	W =    47.745 deg,	P =     8.599 deg,	R =   -35.895 deg
   GP2:
	UF : 1, UT : 1,
	J1=     0.000 deg,	J2=   180.000 deg
};
P[182]{
   GP1:
	UF : 1, UT : 1,		CONFIG : 'N U T, 0, 0, 0',
	X =  2150.796  mm,	Y =    51.228  mm,	Z =   379.826  mm,
	W =     9.396 deg,	P =    -3.028 deg,	R =   -24.284 deg
   GP2:
	UF : 1, UT : 1,
	J1=     0.000 deg,	J2=   180.000 deg
};
P[183]{
   GP1:
	UF : 1, UT : 1,		CONFIG : 'N U T, 0, 0, 0',
	X =  1058.698  mm,	Y =   195.065  mm,	Z =  1283.367  mm,
	W =    73.635 deg,	P =    26.735 deg,	R =   -73.196 deg
   GP2:
	UF : 1, UT : 1,
	J1=   -90.000 deg,	J2=   -90.000 deg
};
P[184]{
   GP1:
	UF : 1, UT : 1,		CONFIG : 'N U T, 0, 0, 0',
	X =  2161.838  mm,	Y =  -354.344  mm,	Z =   373.103  mm,
	W =   -42.503 deg,	P =    -2.383 deg,	R =   -32.742 deg
   GP2:
	UF : 1, UT : 1,
	J1=     0.000 deg,	J2=   180.000 deg
};
P[185]{
   GP1:
	UF : 1, UT : 1,		CONFIG : 'N U T, 0, 0, 0',
	X =  2732.660  mm,	Y =  -291.498  mm,	Z =   459.463  mm,
	W =    29.147 deg,	P =    30.453 deg,	R =  -132.266 deg
   GP2:
	UF : 1, UT : 1,
	J1=    90.000 deg,	J2=     0.000 deg
};
P[186]{
   GP1:
	UF : 1, UT : 1,		CONFIG : 'N U T, 0, 0, 1',
	X =  2737.828  mm,	Y =  -335.614  mm,	Z =   459.309  mm,
	W =    29.459 deg,	P =    30.697 deg,	R =  -132.107 deg
   GP2:
	UF : 1, UT : 1,
	J1=    90.000 deg,	J2=     0.000 deg
};
P[187]{
   GP1:
	UF : 1, UT : 1,		CONFIG : 'N U T, 0, 0, 1',
	X =  2748.682  mm,	Y =  -359.447  mm,	Z =   458.247  mm,
	W =    32.708 deg,	P =    26.756 deg,	R =  -103.211 deg
   GP2:
	UF : 1, UT : 1,
	J1=    90.000 deg,	J2=     0.000 deg
};
P[188]{
   GP1:
	UF : 1, UT : 1,		CONFIG : 'N U T, 0, 0, 1',
	X =  2782.788  mm,	Y =  -368.053  mm,	Z =   461.277  mm,
	W =    32.871 deg,	P =    19.630 deg,	R =   -83.146 deg
   GP2:
	UF : 1, UT : 1,
	J1=    90.000 deg,	J2=     0.000 deg
};
P[189]{
   GP1:
	UF : 1, UT : 1,		CONFIG : 'N U T, 0, 0, 0',
	X =  2149.286  mm,	Y =  -279.133  mm,	Z =   456.472  mm,
	W =   -44.186 deg,	P =    -9.562 deg,	R =     3.909 deg
   GP2:
	UF : 1, UT : 1,
	J1=     0.000 deg,	J2=   180.000 deg
};
P[190]{
   GP1:
	UF : 1, UT : 1,		CONFIG : 'N U T, 0, 0, 1',
	X =  1982.724  mm,	Y =   -25.313  mm,	Z =   235.548  mm,
	W =    21.889 deg,	P =    35.316 deg,	R =  -145.925 deg
   GP2:
	UF : 1, UT : 1,
	J1=     0.000 deg,	J2=   180.000 deg
};
P[191]{
   GP1:
	UF : 1, UT : 1,		CONFIG : 'N U T, 0, 0, 1',
	X =  2182.725  mm,	Y =  -216.312  mm,	Z =    -6.136  mm,
	W =    32.857 deg,	P =    25.665 deg,	R =  -124.570 deg
   GP2:
	UF : 1, UT : 1,
	J1=     0.000 deg,	J2=   180.000 deg
};
P[192]{
   GP1:
	UF : 1, UT : 1,		CONFIG : 'N U T, 0, 0, 0',
	X =  2740.807  mm,	Y =   282.456  mm,	Z =   454.339  mm,
	W =   -36.614 deg,	P =    28.247 deg,	R =   122.490 deg
   GP2:
	UF : 1, UT : 1,
	J1=    90.000 deg,	J2=     0.000 deg
};
P[193]{
   GP1:
	UF : 1, UT : 1,		CONFIG : 'N U T, 0, 0, 0',
	X =  2740.471  mm,	Y =   330.671  mm,	Z =   455.272  mm,
	W =   -36.614 deg,	P =    28.247 deg,	R =   122.490 deg
   GP2:
	UF : 1, UT : 1,
	J1=    90.000 deg,	J2=     0.000 deg
};
P[194]{
   GP1:
	UF : 1, UT : 1,		CONFIG : 'N U T, 0, 0, 0',
	X =  2760.137  mm,	Y =   356.906  mm,	Z =   456.179  mm,
	W =   -32.204 deg,	P =    27.169 deg,	R =   100.051 deg
   GP2:
	UF : 1, UT : 1,
	J1=    90.000 deg,	J2=     0.000 deg
};
P[195]{
   GP1:
	UF : 1, UT : 1,		CONFIG : 'N U T, 0, 0, 1',
	X =  2185.038  mm,	Y =   -47.631  mm,	Z =   -82.880  mm,
	W =     1.218 deg,	P =    44.987 deg,	R =  -147.433 deg
   GP2:
	UF : 1, UT : 1,
	J1=     0.000 deg,	J2=   180.000 deg
};
P[196]{
   GP1:
	UF : 1, UT : 1,		CONFIG : 'N U T, 0, 0, 0',
	X =  2185.038  mm,	Y =   213.369  mm,	Z =   -82.880  mm,
	W =   -26.253 deg,	P =    37.378 deg,	R =   139.534 deg
   GP2:
	UF : 1, UT : 1,
	J1=     0.000 deg,	J2=   180.000 deg
};
P[197]{
   GP1:
	UF : 1, UT : 1,		CONFIG : 'N U T, 0, 0, 0',
	X =  2776.222  mm,	Y =   360.760  mm,	Z =   461.623  mm,
	W =   -28.646 deg,	P =    22.121 deg,	R =    94.724 deg
   GP2:
	UF : 1, UT : 1,
	J1=    90.000 deg,	J2=     0.000 deg
};
P[198]{
   GP1:
	UF : 1, UT : 1,		CONFIG : 'N U T, 0, 0, 0',
	X =  1666.073  mm,	Y =   232.940  mm,	Z =   357.763  mm,
	W =    31.327 deg,	P =    33.496 deg,	R =    49.952 deg
   GP2:
	UF : 1, UT : 1,
	J1=    90.000 deg,	J2=     0.000 deg
};
P[199]{
   GP1:
	UF : 1, UT : 1,		CONFIG : 'N U T, 0, 0, 0',
	X =  1669.367  mm,	Y =   161.118  mm,	Z =   359.810  mm,
	W =    31.331 deg,	P =    33.498 deg,	R =    49.952 deg
   GP2:
	UF : 1, UT : 1,
	J1=    90.000 deg,	J2=     0.000 deg
};
P[200]{
   GP1:
	UF : 1, UT : 1,		CONFIG : 'N U T, 0, 0, 0',
	X =  2149.428  mm,	Y =    61.346  mm,	Z =   -40.697  mm,
	W =    14.710 deg,	P =    43.024 deg,	R =   172.922 deg
   GP2:
	UF : 1, UT : 1,
	J1=     0.000 deg,	J2=   180.000 deg
};
P[201]{
   GP1:
	UF : 1, UT : 1,		CONFIG : 'N U T, 0, 0, 0',
	X =  1379.179  mm,	Y =     5.048  mm,	Z =   295.119  mm,
	W =    -2.053 deg,	P =    45.296 deg,	R =  -168.776 deg
   GP2:
	UF : 1, UT : 1,
	J1=     0.000 deg,	J2=   180.000 deg
};
P[202]{
   GP1:
	UF : 1, UT : 1,		CONFIG : 'N U T, 0, 0, 1',
	X =  1381.432  mm,	Y =  -574.038  mm,	Z =   156.436  mm,
	W =    42.351 deg,	P =    16.902 deg,	R =  -106.783 deg
   GP2:
	UF : 1, UT : 1,
	J1=     0.000 deg,	J2=   180.000 deg
};
P[203]{
   GP1:
	UF : 1, UT : 1,		CONFIG : 'N U T, 0, 0, 0',
	X =  1672.296  mm,	Y =  -245.157  mm,	Z =   359.474  mm,
	W =   -34.074 deg,	P =    31.387 deg,	R =   -56.109 deg
   GP2:
	UF : 1, UT : 1,
	J1=    90.000 deg,	J2=     0.000 deg
};
P[204]{
   GP1:
	UF : 1, UT : 1,		CONFIG : 'N U T, 0, 0, 0',
	X =  1674.067  mm,	Y =  -171.272  mm,	Z =   358.368  mm,
	W =   -34.074 deg,	P =    31.387 deg,	R =   -56.109 deg
   GP2:
	UF : 1, UT : 1,
	J1=    90.000 deg,	J2=     0.000 deg
};
P[205]{
   GP1:
	UF : 1, UT : 1,		CONFIG : 'N U T, 0, 0, 0',
	X =  1806.951  mm,	Y =  -401.301  mm,	Z =   820.124  mm,
	W =     -.611 deg,	P =      .925 deg,	R =   -33.342 deg
   GP2:
	UF : 1, UT : 1,
	J1=    45.000 deg,	J2=     0.000 deg
};
P[206]{
   GP1:
	UF : 1, UT : 1,		CONFIG : 'N U T, 0, 0, 1',
	X =  1351.612  mm,	Y =  -644.118  mm,	Z =   196.361  mm,
	W =    42.489 deg,	P =    16.481 deg,	R =  -107.209 deg
   GP2:
	UF : 1, UT : 1,
	J1=     0.000 deg,	J2=   180.000 deg
};
P[207]{
   GP1:
	UF : 1, UT : 1,		CONFIG : 'N U T, 0, 0, 0',
	X =  1351.612  mm,	Y =     1.774  mm,	Z =   196.362  mm,
	W =     -.786 deg,	P =    44.995 deg,	R =   178.888 deg
   GP2:
	UF : 1, UT : 1,
	J1=     0.000 deg,	J2=   180.000 deg
};
P[208]{
   GP1:
	UF : 1, UT : 1,		CONFIG : 'N U T, 0, 0, 0',
	X =  1811.177  mm,	Y =  -171.928  mm,	Z =   822.372  mm,
	W =     -.615 deg,	P =      .929 deg,	R =   -33.344 deg
   GP2:
	UF : 1, UT : 1,
	J1=    45.000 deg,	J2=     0.000 deg
};
P[209]{
   GP1:
	UF : 1, UT : 1,		CONFIG : 'N U T, 0, 0, 0',
	X =  1807.900  mm,	Y =   392.843  mm,	Z =   821.281  mm,
	W =     -.607 deg,	P =      .924 deg,	R =    40.442 deg
   GP2:
	UF : 1, UT : 1,
	J1=    45.000 deg,	J2=     0.000 deg
};
P[210]{
   GP1:
	UF : 1, UT : 1,		CONFIG : 'N U T, 0, 0, 0',
	X =  1404.034  mm,	Y =  -379.314  mm,	Z =   119.254  mm,
	W =    18.566 deg,	P =    41.762 deg,	R =  -153.239 deg
   GP2:
	UF : 1, UT : 1,
	J1=     0.000 deg,	J2=   180.000 deg
};
P[211]{
   GP1:
	UF : 1, UT : 1,		CONFIG : 'N U T, 0, 0, 0',
	X =  1404.034  mm,	Y =   331.497  mm,	Z =   119.254  mm,
	W =   -20.958 deg,	P =    40.782 deg,	R =   149.612 deg
   GP2:
	UF : 1, UT : 1,
	J1=     0.000 deg,	J2=   180.000 deg
};
P[212]{
   GP1:
	UF : 1, UT : 1,		CONFIG : 'N U T, 0, 0, 0',
	X =  1805.706  mm,	Y =   162.058  mm,	Z =   821.772  mm,
	W =     -.607 deg,	P =      .924 deg,	R =    40.442 deg
   GP2:
	UF : 1, UT : 1,
	J1=    45.000 deg,	J2=     0.000 deg
};
P[213]{
   GP1:
	UF : 1, UT : 1,		CONFIG : 'N U T, 0, 0, 0',
	X =  2179.485  mm,	Y =   641.712  mm,	Z =  1313.269  mm,
	W =     -.150 deg,	P =     3.186 deg,	R =     -.120 deg
   GP2:
	UF : 1, UT : 1,
	J1=   124.996 deg,	J2=     0.000 deg
};
P[214]{
   GP1:
	UF : 1, UT : 1,		CONFIG : 'N U T, 0, 0, 0',
	X =  1267.764  mm,	Y =    -5.079  mm,	Z =   257.741  mm,
	W =     -.786 deg,	P =    44.995 deg,	R =   178.888 deg
   GP2:
	UF : 1, UT : 1,
	J1=     0.000 deg,	J2=   180.000 deg
};
P[215]{
   GP1:
	UF : 1, UT : 1,		CONFIG : 'N U T, 0, 0, 0',
	X =  1267.763  mm,	Y =   567.064  mm,	Z =   257.741  mm,
	W =    24.666 deg,	P =    38.913 deg,	R =  -143.830 deg
   GP2:
	UF : 1, UT : 1,
	J1=     0.000 deg,	J2=   180.000 deg
};
P[216]{
   GP1:
	UF : 1, UT : 1,		CONFIG : 'N U T, 0, 0, 0',
	X =  2180.448  mm,	Y =   484.330  mm,	Z =  1313.381  mm,
	W =      .050 deg,	P =     3.285 deg,	R =     -.057 deg
   GP2:
	UF : 1, UT : 1,
	J1=   124.995 deg,	J2=     0.000 deg
};
P[217]{
   GP1:
	UF : 1, UT : 1,		CONFIG : 'N U T, 0, 0, 0',
	X =  2180.629  mm,	Y =   441.870  mm,	Z =  1314.110  mm,
	W =   -10.967 deg,	P =     3.763 deg,	R =     -.257 deg
   GP2:
	UF : 1, UT : 1,
	J1=   124.999 deg,	J2=     0.000 deg
};
P[218]{
   GP1:
	UF : 1, UT : 1,		CONFIG : 'N U T, 0, 0, 0',
	X =  2166.448  mm,	Y =     9.539  mm,	Z =  1331.644  mm,
	W =     -.712 deg,	P =     8.094 deg,	R =     -.112 deg
   GP2:
	UF : 1, UT : 1,
	J1=   124.996 deg,	J2=     0.000 deg
};
P[219]{
   GP1:
	UF : 1, UT : 1,		CONFIG : 'N U T, 0, 0, 0',
	X =  1302.181  mm,	Y =   638.659  mm,	Z =   248.465  mm,
	W =    31.136 deg,	P =    34.298 deg,	R =  -133.008 deg
   GP2:
	UF : 1, UT : 1,
	J1=     0.000 deg,	J2=   180.000 deg
};
P[220]{
   GP1:
	UF : 1, UT : 1,		CONFIG : 'N U T, 0, 0, 0',
	X =  1186.272  mm,	Y =   472.511  mm,	Z =   672.833  mm,
	W =    32.440 deg,	P =    45.276 deg,	R =   -70.624 deg
   GP2:
	UF : 1, UT : 1,
	J1=     0.000 deg,	J2=   180.000 deg
};
P[221]{
   GP1:
	UF : 1, UT : 1,		CONFIG : 'N U T, 0, 0, 0',
	X =  2166.019  mm,	Y =  -184.522  mm,	Z =  1332.900  mm,
	W =     -.016 deg,	P =    10.106 deg,	R =      .980 deg
   GP2:
	UF : 1, UT : 1,
	J1=   125.000 deg,	J2=     0.000 deg
};
P[222]{
   GP1:
	UF : 1, UT : 1,		CONFIG : 'N U T, 0, 0, 0',
	X =  2166.456  mm,	Y =  -407.129  mm,	Z =  1331.643  mm,
	W =     -.927 deg,	P =     7.509 deg,	R =     -.098 deg
   GP2:
	UF : 1, UT : 1,
	J1=   125.000 deg,	J2=     0.000 deg
};
P[223]{
   GP1:
	UF : 1, UT : 1,		CONFIG : 'N U T, 0, 0, 0',
	X =  2167.632  mm,	Y =   399.347  mm,	Z =  1331.502  mm,
	W =      .164 deg,	P =     6.215 deg,	R =      .006 deg
   GP2:
	UF : 1, UT : 1,
	J1=   125.000 deg,	J2=     0.000 deg
};
P[224]{
   GP1:
	UF : 1, UT : 1,		CONFIG : 'N U T, 0, 0, 0',
	X =  1759.654  mm,	Y =  1128.978  mm,	Z =   266.859  mm,
	W =   -16.763 deg,	P =    16.253 deg,	R =    47.184 deg
   GP2:
	UF : 1, UT : 1,
	J1=    90.000 deg,	J2=    90.000 deg
};
P[225]{
   GP1:
	UF : 1, UT : 1,		CONFIG : 'N U T, 0, 0, 0',
	X =  1547.891  mm,	Y =   -77.836  mm,	Z =    80.464  mm,
	W =     5.459 deg,	P =    -9.689 deg,	R =   -27.215 deg
   GP2:
	UF : 1, UT : 1,
	J1=     0.000 deg,	J2=   180.000 deg
};
P[226]{
   GP1:
	UF : 1, UT : 1,		CONFIG : 'N U T, 0, 0, 0',
	X =  2166.862  mm,	Y =   175.690  mm,	Z =  1332.608  mm,
	W =      .990 deg,	P =     7.423 deg,	R =      .117 deg
   GP2:
	UF : 1, UT : 1,
	J1=   125.000 deg,	J2=     0.000 deg
};
P[227]{
   GP1:
	UF : 1, UT : 1,		CONFIG : 'N U T, 0, 0, 0',
	X =  2166.171  mm,	Y =     8.099  mm,	Z =  1332.684  mm,
	W =    -1.725 deg,	P =     7.606 deg,	R =     2.359 deg
   GP2:
	UF : 1, UT : 1,
	J1=   125.000 deg,	J2=     0.000 deg
};
P[228]{
   GP1:
	UF : 1, UT : 1,		CONFIG : 'N U T, 0, 0, 0',
	X =  2179.486  mm,	Y =  -651.866  mm,	Z =  1318.869  mm,
	W =      .005 deg,	P =     8.099 deg,	R =      .006 deg
   GP2:
	UF : 1, UT : 1,
	J1=   125.000 deg,	J2=     0.000 deg
};
P[229]{
   GP1:
	UF : 1, UT : 1,		CONFIG : 'N U T, 0, 0, 0',
	X =  2179.374  mm,	Y =  -454.527  mm,	Z =  1315.208  mm,
	W =      .023 deg,	P =     7.896 deg,	R =     -.019 deg
   GP2:
	UF : 1, UT : 1,
	J1=   125.000 deg,	J2=     0.000 deg
};
P[230]{
   GP1:
	UF : 1, UT : 1,		CONFIG : 'N U T, 0, 0, 0',
	X =  1458.812  mm,	Y =  -160.809  mm,	Z =   231.788  mm,
	W =     9.627 deg,	P =   -18.262 deg,	R =   -28.428 deg
   GP2:
	UF : 1, UT : 1,
	J1=     0.000 deg,	J2=   180.000 deg
};
P[231]{
   GP1:
	UF : 1, UT : 1,		CONFIG : 'N U T, 0, 0, 0',
	X =  2179.713  mm,	Y =  -448.929  mm,	Z =  1315.415  mm,
	W =     8.588 deg,	P =     5.688 deg,	R =      .847 deg
   GP2:
	UF : 1, UT : 1,
	J1=   125.000 deg,	J2=     0.000 deg
};
P[232]{
   GP1:
	UF : 1, UT : 1,		CONFIG : 'N U T, 0, 0, 0',
	X =  2140.306  mm,	Y =   407.443  mm,	Z =   274.579  mm,
	W =    39.266 deg,	P =    23.844 deg,	R =     9.200 deg
   GP2:
	UF : 1, UT : 1,
	J1=     0.000 deg,	J2=   180.000 deg
};
P[233]{
   GP1:
	UF : 1, UT : 1,		CONFIG : 'N U T, 0, 0, 0',
	X =  2171.990  mm,	Y =   -24.925  mm,	Z =  -336.558  mm,
	W =    -4.854 deg,	P =     4.648 deg,	R =    10.738 deg
   GP2:
	UF : 1, UT : 1,
	J1=    45.000 deg,	J2=   182.246 deg
};
P[234]{
   GP1:
	UF : 1, UT : 1,		CONFIG : 'N U T, 0, 0, 0',
	X =  2525.957  mm,	Y =  -153.860  mm,	Z =   104.179  mm,
	W =    36.503 deg,	P =    18.679 deg,	R =   -19.970 deg
   GP2:
	UF : 1, UT : 1,
	J1=    80.000 deg,	J2=    90.000 deg
};
P[235]{
   GP1:
	UF : 1, UT : 1,		CONFIG : 'N U T, 0, 0, 0',
	X =  2443.957  mm,	Y =  -153.860  mm,	Z =    41.179  mm,
	W =    36.503 deg,	P =    18.679 deg,	R =    32.647 deg
   GP2:
	UF : 1, UT : 1,
	J1=    80.000 deg,	J2=    90.000 deg
};
P[236]{
   GP1:
	UF : 1, UT : 1,		CONFIG : 'N U T, 0, 0, 0',
	X =  2156.848  mm,	Y =   408.546  mm,	Z =   273.021  mm,
	W =    39.276 deg,	P =    23.852 deg,	R =   -24.752 deg
   GP2:
	UF : 1, UT : 1,
	J1=     0.000 deg,	J2=   180.000 deg
};
P[237]{
   GP1:
	UF : 1, UT : 1,		CONFIG : 'N U T, 0, 0, 0',
	X =  2192.264  mm,	Y =   408.269  mm,	Z =   272.683  mm,
	W =    39.348 deg,	P =    23.574 deg,	R =   -24.954 deg
   GP2:
	UF : 1, UT : 1,
	J1=     0.000 deg,	J2=   180.000 deg
};
P[238]{
   GP1:
	UF : 1, UT : 1,		CONFIG : 'N U T, 0, 0, 0',
	X =  2195.713  mm,	Y =   409.133  mm,	Z =   275.050  mm,
	W =    41.358 deg,	P =    16.787 deg,	R =   -30.152 deg
   GP2:
	UF : 1, UT : 1,
	J1=     0.000 deg,	J2=   180.000 deg
};
P[239]{
   GP1:
	UF : 1, UT : 1,		CONFIG : 'N U T, 0, 0, 0',
	X =  2131.308  mm,	Y =  -414.633  mm,	Z =   275.688  mm,
	W =   -42.902 deg,	P =    -2.083 deg,	R =   -37.986 deg
   GP2:
	UF : 1, UT : 1,
	J1=     0.000 deg,	J2=   180.000 deg
};
P[240]{
   GP1:
	UF : 1, UT : 1,		CONFIG : 'N U T, 0, 0, 0',
	X =  2443.958  mm,	Y =  -141.290  mm,	Z =    41.179  mm,
	W =    36.502 deg,	P =    18.679 deg,	R =    44.252 deg
   GP2:
	UF : 1, UT : 1,
	J1=    80.000 deg,	J2=    90.000 deg
};
P[241]{
   GP1:
	UF : 1, UT : 1,		CONFIG : 'N U T, 0, 0, 0',
	X =  2525.957  mm,	Y =  -153.860  mm,	Z =   104.179  mm,
	W =    36.503 deg,	P =    18.679 deg,	R =   -19.970 deg
   GP2:
	UF : 1, UT : 1,
	J1=    80.000 deg,	J2=    90.000 deg
};
P[242]{
   GP1:
	UF : 1, UT : 1,		CONFIG : 'N U T, 0, 0, 0',
	X =  1638.942  mm,	Y =  -220.932  mm,	Z =   176.092  mm,
	W =    39.659 deg,	P =    20.135 deg,	R =   -30.806 deg
   GP2:
	UF : 1, UT : 1,
	J1=    90.000 deg,	J2=    90.000 deg
};
P[243]{
   GP1:
	UF : 1, UT : 1,		CONFIG : 'N U T, 0, 0, 0',
	X =  1677.355  mm,	Y =  -241.647  mm,	Z =    77.021  mm,
	W =    39.659 deg,	P =    20.135 deg,	R =   -14.061 deg
   GP2:
	UF : 1, UT : 1,
	J1=    90.000 deg,	J2=    90.000 deg
};
P[244]{
   GP1:
	UF : 1, UT : 1,		CONFIG : 'N U T, 0, 0, 0',
	X =  2148.323  mm,	Y =  -414.723  mm,	Z =   274.084  mm,
	W =   -42.900 deg,	P =    -2.086 deg,	R =    -3.516 deg
   GP2:
	UF : 1, UT : 1,
	J1=     0.000 deg,	J2=   180.000 deg
};
P[245]{
   GP1:
	UF : 1, UT : 1,		CONFIG : 'N U T, 0, 0, 0',
	X =  2197.502  mm,	Y =  -415.369  mm,	Z =   273.507  mm,
	W =   -42.900 deg,	P =    -2.086 deg,	R =    -3.516 deg
   GP2:
	UF : 1, UT : 1,
	J1=     0.000 deg,	J2=   180.000 deg
};
P[246]{
   GP1:
	UF : 1, UT : 1,		CONFIG : 'N U T, 0, 0, 0',
	X =  2205.828  mm,	Y =  -413.909  mm,	Z =   275.461  mm,
	W =   -37.675 deg,	P =   -22.312 deg,	R =     8.930 deg
   GP2:
	UF : 1, UT : 1,
	J1=     0.000 deg,	J2=   180.000 deg
};
P[247]{
   GP1:
	UF : 1, UT : 1,		CONFIG : 'N U T, 0, 0, 1',
	X =  2230.692  mm,	Y =  -244.712  mm,	Z =  -195.164  mm,
	W =    34.818 deg,	P =    27.072 deg,	R =  -123.443 deg
   GP2:
	UF : 1, UT : 1,
	J1=     0.000 deg,	J2=   180.000 deg
};
P[248]{
   GP1:
	UF : 1, UT : 1,		CONFIG : 'N U T, 0, 0, 0',
	X =  1961.011  mm,	Y =  -250.911  mm,	Z =    63.963  mm,
	W =    38.570 deg,	P =    15.643 deg,	R =   -37.733 deg
   GP2:
	UF : 1, UT : 1,
	J1=    90.000 deg,	J2=    90.000 deg
};
P[249]{
   GP1:
	UF : 1, UT : 1,		CONFIG : 'N U T, 0, 0, 0',
	X =  2227.011  mm,	Y =   -35.911  mm,	Z =    63.963  mm,
	W =    41.142 deg,	P =     1.290 deg,	R =    -4.650 deg
   GP2:
	UF : 1, UT : 1,
	J1=    90.000 deg,	J2=    90.000 deg
};
P[250]{
   GP1:
	UF : 1, UT : 1,		CONFIG : 'N U T, 0, 0, 1',
	X =  2231.573  mm,	Y =   -26.230  mm,	Z =  -195.203  mm,
	W =    34.826 deg,	P =    27.077 deg,	R =  -123.454 deg
   GP2:
	UF : 1, UT : 1,
	J1=     0.000 deg,	J2=   180.000 deg
};
P[251]{
   GP1:
	UF : 1, UT : 1,		CONFIG : 'N U T, 0, 0, 1',
	X =  2228.732  mm,	Y =    -5.925  mm,	Z =  -190.893  mm,
	W =    33.017 deg,	P =    26.717 deg,	R =   -93.421 deg
   GP2:
	UF : 1, UT : 1,
	J1=     0.000 deg,	J2=   180.000 deg
};
P[252]{
   GP1:
	UF : 1, UT : 1,		CONFIG : 'N U T, 0, 0, 0',
	X =  2193.552  mm,	Y =   -35.911  mm,	Z =    63.963  mm,
	W =    41.142 deg,	P =     1.290 deg,	R =    -4.650 deg
   GP2:
	UF : 1, UT : 1,
	J1=    90.000 deg,	J2=    90.000 deg
};
P[253]{
   GP1:
	UF : 1, UT : 1,		CONFIG : 'N U T, 0, 0, 0',
	X =  2230.608  mm,	Y =   237.638  mm,	Z =  -198.866  mm,
	W =   -26.756 deg,	P =    37.336 deg,	R =   139.554 deg
   GP2:
	UF : 1, UT : 1,
	J1=     0.000 deg,	J2=   180.000 deg
};
P[254]{
   GP1:
	UF : 1, UT : 1,		CONFIG : 'N U T, 0, 0, 0',
	X =  2230.167  mm,	Y =    15.957  mm,	Z =  -196.509  mm,
	W =   -26.754 deg,	P =    37.334 deg,	R =   139.553 deg
   GP2:
	UF : 1, UT : 1,
	J1=     0.000 deg,	J2=   180.000 deg
};
P[255]{
   GP1:
	UF : 1, UT : 1,		CONFIG : 'N U T, 0, 0, 0',
	X =  2229.296  mm,	Y =    -3.861  mm,	Z =  -195.798  mm,
	W =   -20.120 deg,	P =    35.519 deg,	R =   111.508 deg
   GP2:
	UF : 1, UT : 1,
	J1=     0.000 deg,	J2=   180.000 deg
};
P[256]{
   GP1:
	UF : 1, UT : 1,		CONFIG : 'N U T, 0, 0, 0',
	X =  2104.646  mm,	Y =   -14.305  mm,	Z =    58.276  mm,
	W =    44.920 deg,	P =     3.025 deg,	R =    -3.029 deg
   GP2:
	UF : 1, UT : 1,
	J1=    90.000 deg,	J2=    90.000 deg
};
P[257]{
   GP1:
	UF : 1, UT : 1,		CONFIG : 'N U T, 0, 0, 0',
	X =  1481.773  mm,	Y =  -649.516  mm,	Z =     4.672  mm,
	W =    42.305 deg,	P =    16.820 deg,	R =  -100.938 deg
   GP2:
	UF : 1, UT : 1,
	J1=     0.000 deg,	J2=   180.000 deg
};
P[258]{
   GP1:
	UF : 1, UT : 1,		CONFIG : 'N U T, 0, 0, 0',
	X =  1483.359  mm,	Y =  -463.806  mm,	Z =     3.440  mm,
	W =    42.353 deg,	P =    16.915 deg,	R =  -100.930 deg
   GP2:
	UF : 1, UT : 1,
	J1=     0.000 deg,	J2=   180.000 deg
};
P[259]{
   GP1:
	UF : 1, UT : 1,		CONFIG : 'N U T, 0, 0, 1',
	X =  1480.083  mm,	Y =  -453.844  mm,	Z =     3.901  mm,
	W =    42.350 deg,	P =    16.901 deg,	R =   -86.937 deg
   GP2:
	UF : 1, UT : 1,
	J1=     0.000 deg,	J2=   180.000 deg
};
P[260]{
   GP1:
	UF : 1, UT : 1,		CONFIG : 'N U T, 0, 0, 0',
	X =  2104.646  mm,	Y =   -54.652  mm,	Z =   175.276  mm,
	W =    44.920 deg,	P =     3.025 deg,	R =    -3.029 deg
   GP2:
	UF : 1, UT : 1,
	J1=    90.000 deg,	J2=    90.000 deg
};
P[261]{
   GP1:
	UF : 1, UT : 1,		CONFIG : 'N U T, 0, 0, 0',
	X =  1705.582  mm,	Y =   -41.652  mm,	Z =   107.776  mm,
	W =    44.920 deg,	P =     3.025 deg,	R =    11.940 deg
   GP2:
	UF : 1, UT : 1,
	J1=    90.000 deg,	J2=    90.000 deg
};
P[262]{
   GP1:
	UF : 1, UT : 1,		CONFIG : 'N U T, 0, 0, -1',
	X =  1457.610  mm,	Y =    -5.074  mm,	Z =    -1.334  mm,
	W =      .944 deg,	P =    42.924 deg,	R =   177.949 deg
   GP2:
	UF : 1, UT : 1,
	J1=     0.000 deg,	J2=   180.000 deg
};
P[263]{
   GP1:
	UF : 1, UT : 1,		CONFIG : 'N U T, 0, 0, 0',
	X =  1456.823  mm,	Y =  -333.215  mm,	Z =     -.642  mm,
	W =    -1.375 deg,	P =    43.930 deg,	R =   175.836 deg
   GP2:
	UF : 1, UT : 1,
	J1=     0.000 deg,	J2=   180.000 deg
};
P[264]{
   GP1:
	UF : 1, UT : 1,		CONFIG : 'N U T, 0, 0, 0',
	X =  1457.144  mm,	Y =  -389.993  mm,	Z =      .340  mm,
	W =     5.164 deg,	P =    43.292 deg,	R =  -179.576 deg
   GP2:
	UF : 1, UT : 1,
	J1=     0.000 deg,	J2=   180.000 deg
};
P[265]{
   GP1:
	UF : 1, UT : 1,		CONFIG : 'N U T, 0, 0, 0',
	X =  1700.208  mm,	Y =   -40.379  mm,	Z =   119.303  mm,
	W =    53.172 deg,	P =     1.611 deg,	R =    24.177 deg
   GP2:
	UF : 1, UT : 1,
	J1=    90.000 deg,	J2=    90.000 deg
};
P[266]{
   GP1:
	UF : 1, UT : 1,		CONFIG : 'N U T, 0, 0, -1',
	X =  1452.091  mm,	Y =   380.184  mm,	Z =     1.132  mm,
	W =    -1.242 deg,	P =    44.316 deg,	R =   179.193 deg
   GP2:
	UF : 1, UT : 1,
	J1=     0.000 deg,	J2=   180.000 deg
};
P[267]{
   GP1:
	UF : 1, UT : 1,		CONFIG : 'N U T, 0, 0, 0',
	X =  1459.905  mm,	Y =    -8.182  mm,	Z =     -.258  mm,
	W =     -.052 deg,	P =    43.981 deg,	R =  -179.147 deg
   GP2:
	UF : 1, UT : 1,
	J1=     0.000 deg,	J2=   180.000 deg
};
P[268]{
   GP1:
	UF : 1, UT : 1,		CONFIG : 'N U T, 0, 0, 0',
	X =  1478.049  mm,	Y =   642.654  mm,	Z =     4.653  mm,
	W =    29.663 deg,	P =    31.501 deg,	R =  -136.780 deg
   GP2:
	UF : 1, UT : 1,
	J1=     0.000 deg,	J2=   180.000 deg
};
P[269]{
   GP1:
	UF : 1, UT : 1,		CONFIG : 'N U T, 0, 0, 0',
	X =  1902.999  mm,	Y =   -46.261  mm,	Z =   175.051  mm,
	W =    52.365 deg,	P =    -4.474 deg,	R =   -14.021 deg
   GP2:
	UF : 1, UT : 1,
	J1=    90.000 deg,	J2=    90.000 deg
};
P[270]{
   GP1:
	UF : 1, UT : 1,		CONFIG : 'N U T, 0, 0, 0',
	X =  1161.856  mm,	Y =   -92.689  mm,	Z =   175.051  mm,
	W =    38.130 deg,	P =    -5.720 deg,	R =    -4.359 deg
   GP2:
	UF : 1, UT : 1,
	J1=    90.000 deg,	J2=    90.000 deg
};
P[271]{
   GP1:
	UF : 1, UT : 1,		CONFIG : 'N U T, 0, 0, 0',
	X =  1353.427  mm,	Y =   457.025  mm,	Z =   417.051  mm,
	W =    -2.563 deg,	P =     5.520 deg,	R =     2.347 deg
   GP2:
	UF : 1, UT : 1,
	J1=    90.000 deg,	J2=    90.000 deg
};
P[272]{
   GP1:
	UF : 1, UT : 1,		CONFIG : 'N U T, 0, 0, 0',
	X =  1530.428  mm,	Y =   623.025  mm,	Z =   175.051  mm,
	W =   -41.304 deg,	P =     5.776 deg,	R =    -1.616 deg
   GP2:
	UF : 1, UT : 1,
	J1=    90.000 deg,	J2=    90.000 deg
};
P[273]{
   GP1:
	UF : 1, UT : 1,		CONFIG : 'N U T, 0, 0, 0',
	X =  2221.857  mm,	Y =   134.025  mm,	Z =   133.501  mm,
	W =   -39.814 deg,	P =   -13.337 deg,	R =   -23.619 deg
   GP2:
	UF : 1, UT : 1,
	J1=    90.000 deg,	J2=    90.000 deg
};
P[274]{
   GP1:
	UF : 1, UT : 1,		CONFIG : 'N U T, 0, 0, 0',
	X =  1475.653  mm,	Y =   450.274  mm,	Z =     6.255  mm,
	W =    35.513 deg,	P =    24.469 deg,	R =  -124.378 deg
   GP2:
	UF : 1, UT : 1,
	J1=     0.000 deg,	J2=   180.000 deg
};
P[275]{
   GP1:
	UF : 1, UT : 1,		CONFIG : 'N U T, 0, 0, 0',
	X =  1474.914  mm,	Y =   441.895  mm,	Z =     5.846  mm,
	W =    35.513 deg,	P =    24.469 deg,	R =  -129.749 deg
   GP2:
	UF : 1, UT : 1,
	J1=     0.000 deg,	J2=   180.000 deg
};
P[276]{
   GP1:
	UF : 1, UT : 1,		CONFIG : 'N U T, 0, 0, 0',
	X =  2162.665  mm,	Y =   110.242  mm,	Z =    59.358  mm,
	W =   -44.607 deg,	P =    -6.682 deg,	R =    -6.729 deg
   GP2:
	UF : 1, UT : 1,
	J1=    90.000 deg,	J2=    90.000 deg
};
P[277]{
   GP1:
	UF : 1, UT : 1,		CONFIG : 'N U T, 0, 0, 0',
	X =  2186.980  mm,	Y =   -83.076  mm,	Z =  -438.565  mm,
	W =     -.956 deg,	P =    22.926 deg,	R =     1.001 deg
   GP2:
	UF : 1, UT : 1,
	J1=    45.000 deg,	J2=   180.000 deg
};
P[278]{
   GP1:
	UF : 1, UT : 1,		CONFIG : 'N U T, 0, 0, 0',
	X =  2186.499  mm,	Y =  -161.647  mm,	Z =  -438.565  mm,
	W =     -.956 deg,	P =    22.926 deg,	R =    22.592 deg
   GP2:
	UF : 1, UT : 1,
	J1=    45.000 deg,	J2=   180.000 deg
};
P[279]{
   GP1:
	UF : 1, UT : 1,		CONFIG : 'N U T, 0, 0, 0',
	X =  1524.716  mm,	Y =   -79.047  mm,	Z =   -64.180  mm,
	W =     1.172 deg,	P =   -23.208 deg,	R =    -8.280 deg
   GP2:
	UF : 1, UT : 1,
	J1=     0.000 deg,	J2=   180.000 deg
};
P[280]{
   GP1:
	UF : 1, UT : 1,		CONFIG : 'N U T, 0, 0, 0',
	X =  2200.817  mm,	Y =   103.879  mm,	Z =    45.598  mm,
	W =   -44.607 deg,	P =    -6.682 deg,	R =    -6.729 deg
   GP2:
	UF : 1, UT : 1,
	J1=    90.000 deg,	J2=    90.000 deg
};
P[281]{
   GP1:
	UF : 1, UT : 1,		CONFIG : 'N U T, 0, 0, 0',
	X =  1991.025  mm,	Y =   103.879  mm,	Z =    45.598  mm,
	W =   -44.607 deg,	P =    -6.682 deg,	R =    -6.729 deg
   GP2:
	UF : 1, UT : 1,
	J1=    90.000 deg,	J2=    90.000 deg
};
P[282]{
   GP1:
	UF : 1, UT : 1,		CONFIG : 'N U T, 0, 0, 0',
	X =  1525.494  mm,	Y =  -112.165  mm,	Z =   -64.782  mm,
	W =     1.185 deg,	P =   -23.204 deg,	R =    -8.290 deg
   GP2:
	UF : 1, UT : 1,
	J1=     0.000 deg,	J2=   180.000 deg
};
P[283]{
   GP1:
	UF : 1, UT : 1,		CONFIG : 'N U T, 0, 0, 0',
	X =  1525.388  mm,	Y =  -160.517  mm,	Z =   -66.135  mm,
	W =     1.184 deg,	P =   -23.205 deg,	R =    -8.289 deg
   GP2:
	UF : 1, UT : 1,
	J1=     0.000 deg,	J2=   180.000 deg
};
P[284]{
   GP1:
	UF : 1, UT : 1,		CONFIG : 'N U T, 0, 0, 0',
	X =  1526.724  mm,	Y =  -137.443  mm,	Z =   -67.899  mm,
	W =     1.184 deg,	P =   -23.205 deg,	R =    -8.289 deg
   GP2:
	UF : 1, UT : 1,
	J1=     0.000 deg,	J2=   180.000 deg
};
P[285]{
   GP1:
	UF : 1, UT : 1,		CONFIG : 'N U T, 0, 0, 0',
	X =  2086.451  mm,	Y =   114.405  mm,	Z =   133.369  mm,
	W =   -44.606 deg,	P =    -6.682 deg,	R =     6.426 deg
   GP2:
	UF : 1, UT : 1,
	J1=    90.000 deg,	J2=    90.000 deg
};
P[286]{
   GP1:
	UF : 1, UT : 1,		CONFIG : 'N U T, 0, 0, 0',
	X =  2121.394  mm,	Y =   114.404  mm,	Z =   147.283  mm,
	W =   -41.424 deg,	P =   -19.434 deg,	R =   -97.506 deg
   GP2:
	UF : 1, UT : 1,
	J1=    90.000 deg,	J2=   100.000 deg
};
P[287]{
   GP1:
	UF : 1, UT : 1,		CONFIG : 'N U T, 0, 0, 0',
	X =  2080.531  mm,	Y =    -7.596  mm,	Z =    92.282  mm,
	W =   -41.424 deg,	P =   -19.434 deg,	R =   -97.506 deg
   GP2:
	UF : 1, UT : 1,
	J1=    90.000 deg,	J2=   100.000 deg
};
P[288]{
   GP1:
	UF : 1, UT : 1,		CONFIG : 'N U T, 0, 0, 0',
	X =  2372.493  mm,	Y =   -85.125  mm,	Z =   -28.442  mm,
	W =    40.515 deg,	P =    40.131 deg,	R =    23.483 deg
   GP2:
	UF : 1, UT : 1,
	J1=    80.000 deg,	J2=    90.000 deg
};
P[289]{
   GP1:
	UF : 1, UT : 1,		CONFIG : 'N U T, 0, 0, 0',
	X =  2370.298  mm,	Y =  -109.505  mm,	Z =   -29.922  mm,
	W =    40.520 deg,	P =    40.127 deg,	R =    54.928 deg
   GP2:
	UF : 1, UT : 1,
	J1=    80.000 deg,	J2=    90.000 deg
};
P[290]{
   GP1:
	UF : 1, UT : 1,		CONFIG : 'N U T, 0, 0, 0',
	X =  2080.530  mm,	Y =    -7.596  mm,	Z =    92.282  mm,
	W =   -41.424 deg,	P =   -19.434 deg,	R =   -97.506 deg
   GP2:
	UF : 1, UT : 1,
	J1=    90.000 deg,	J2=   100.000 deg
};
P[291]{
   GP1:
	UF : 1, UT : 1,		CONFIG : 'N U T, 0, 0, 0',
	X =  2080.530  mm,	Y =   309.547  mm,	Z =   503.711  mm,
	W =    -3.830 deg,	P =   -10.878 deg,	R =   -17.892 deg
   GP2:
	UF : 1, UT : 1,
	J1=    90.000 deg,	J2=   135.000 deg
};
P[292]{
   GP1:
	UF : 1, UT : 1,		CONFIG : 'N U T, 0, 0, 0',
	X =  2670.559  mm,	Y =   209.547  mm,	Z =   314.711  mm,
	W =    -3.830 deg,	P =   -10.878 deg,	R =   -17.892 deg
   GP2:
	UF : 1, UT : 1,
	J1=    90.000 deg,	J2=   135.000 deg
};
P[293]{
   GP1:
	UF : 1, UT : 1,		CONFIG : 'N U T, 0, 0, 0',
	X =  2373.512  mm,	Y =  -147.571  mm,	Z =   -28.085  mm,
	W =    40.521 deg,	P =    40.128 deg,	R =    54.929 deg
   GP2:
	UF : 1, UT : 1,
	J1=    80.000 deg,	J2=    90.000 deg
};
P[294]{
   GP1:
	UF : 1, UT : 1,		CONFIG : 'N U T, 0, 0, 0',
	X =  2373.382  mm,	Y =  -159.792  mm,	Z =   -26.936  mm,
	W =    39.996 deg,	P =    39.207 deg,	R =    81.747 deg
   GP2:
	UF : 1, UT : 1,
	J1=    79.998 deg,	J2=    90.000 deg
};
P[295]{
   GP1:
	UF : 1, UT : 1,		CONFIG : 'N U T, 0, 0, 0',
	X =  2649.168  mm,	Y =   166.049  mm,	Z =   301.659  mm,
	W =    13.374 deg,	P =   -35.036 deg,	R =   -22.495 deg
   GP2:
	UF : 1, UT : 1,
	J1=    90.000 deg,	J2=   135.000 deg
};
P[296]{
   GP1:
	UF : 1, UT : 1,		CONFIG : 'N U T, 0, 0, 0',
	X =  2349.168  mm,	Y =   281.049  mm,	Z =   301.659  mm,
	W =     -.090 deg,	P =    -5.498 deg,	R =      .950 deg
   GP2:
	UF : 1, UT : 1,
	J1=    90.000 deg,	J2=   135.000 deg
};
P[297]{
   GP1:
	UF : 1, UT : 1,		CONFIG : 'N U T, 0, 0, 0',
	X =  1674.558  mm,	Y =  -197.902  mm,	Z =   -15.747  mm,
	W =    38.571 deg,	P =    15.643 deg,	R =    22.733 deg
   GP2:
	UF : 1, UT : 1,
	J1=    90.000 deg,	J2=    90.000 deg
};
P[298]{
   GP1:
	UF : 1, UT : 1,		CONFIG : 'N U T, 0, 0, 0',
	X =  1706.028  mm,	Y =  -198.510  mm,	Z =   -16.685  mm,
	W =    38.571 deg,	P =    15.644 deg,	R =   -27.579 deg
   GP2:
	UF : 1, UT : 1,
	J1=    90.000 deg,	J2=    90.000 deg
};
P[299]{
   GP1:
	UF : 1, UT : 1,		CONFIG : 'N U T, 0, 0, 0',
	X =  2703.820  mm,	Y =   252.204  mm,	Z =   224.219  mm,
	W =     -.140 deg,	P =    -8.465 deg,	R =      .956 deg
   GP2:
	UF : 1, UT : 1,
	J1=    90.000 deg,	J2=   135.000 deg
};
P[300]{
   GP1:
	UF : 1, UT : 1,		CONFIG : 'N U T, 0, 0, 0',
	X =  2289.178  mm,	Y =   268.490  mm,	Z =   224.220  mm,
	W =     -.140 deg,	P =    -8.465 deg,	R =      .956 deg
   GP2:
	UF : 1, UT : 1,
	J1=    90.000 deg,	J2=   135.000 deg
};
P[301]{
   GP1:
	UF : 1, UT : 1,		CONFIG : 'N U T, 0, 0, 0',
	X =  1843.464  mm,	Y =   431.347  mm,	Z =   609.934  mm,
	W =     -.140 deg,	P =    -8.465 deg,	R =   -19.002 deg
   GP2:
	UF : 1, UT : 1,
	J1=    90.000 deg,	J2=   135.000 deg
};
P[302]{
   GP1:
	UF : 1, UT : 1,		CONFIG : 'N U T, 0, 0, 0',
	X =  1843.464  mm,	Y =   431.347  mm,	Z =   378.506  mm,
	W =    39.110 deg,	P =     2.688 deg,	R =   -82.797 deg
   GP2:
	UF : 1, UT : 1,
	J1=    90.000 deg,	J2=    90.000 deg
};
P[303]{
   GP1:
	UF : 1, UT : 1,		CONFIG : 'N U T, 0, 0, 0',
	X =  2020.464  mm,	Y =   107.456  mm,	Z =   101.505  mm,
	W =    39.110 deg,	P =     2.688 deg,	R =   -82.797 deg
   GP2:
	UF : 1, UT : 1,
	J1=    90.000 deg,	J2=    90.000 deg
};
P[304]{
   GP1:
	UF : 1, UT : 1,		CONFIG : 'N U T, 0, 0, 0',
	X =  1973.574  mm,	Y =  -202.749  mm,	Z =   -17.434  mm,
	W =    38.571 deg,	P =    15.644 deg,	R =   -27.579 deg
   GP2:
	UF : 1, UT : 1,
	J1=    90.000 deg,	J2=    90.000 deg
};
P[305]{
   GP1:
	UF : 1, UT : 1,		CONFIG : 'N U T, 0, 0, 0',
	X =  1991.550  mm,	Y =  -201.914  mm,	Z =   -14.547  mm,
	W =    38.530 deg,	P =    15.652 deg,	R =   -66.405 deg
   GP2:
	UF : 1, UT : 1,
	J1=    89.999 deg,	J2=    90.000 deg
};
P[306]{
   GP1:
	UF : 1, UT : 1,		CONFIG : 'N U T, 0, 0, 0',
	X =  2220.122  mm,	Y =    37.299  mm,	Z =    -4.302  mm,
	W =    44.923 deg,	P =     3.028 deg,	R =    -3.033 deg
   GP2:
	UF : 1, UT : 1,
	J1=    90.000 deg,	J2=    90.000 deg
};
P[307]{
   GP1:
	UF : 1, UT : 1,		CONFIG : 'N U T, 0, 0, -1',
	X =  2012.815  mm,	Y =   114.104  mm,	Z =    90.700  mm,
	W =    40.362 deg,	P =    21.867 deg,	R =  -139.995 deg
   GP2:
	UF : 1, UT : 1,
	J1=    90.000 deg,	J2=    90.000 deg
};
P[308]{
   GP1:
	UF : 1, UT : 1,		CONFIG : 'N U T, 0, 0, 0',
	X =  1644.243  mm,	Y =   456.961  mm,	Z =    90.700  mm,
	W =   -42.959 deg,	P =    14.926 deg,	R =    16.534 deg
   GP2:
	UF : 1, UT : 1,
	J1=    90.000 deg,	J2=    90.000 deg
};
P[309]{
   GP1:
	UF : 1, UT : 1,		CONFIG : 'N U T, 0, 0, 0',
	X =  1667.302  mm,	Y =   122.961  mm,	Z =    90.700  mm,
	W =   -42.959 deg,	P =    14.926 deg,	R =    16.534 deg
   GP2:
	UF : 1, UT : 1,
	J1=    90.000 deg,	J2=    90.000 deg
};
P[310]{
   GP1:
	UF : 1, UT : 1,		CONFIG : 'N U T, 0, 0, 0',
	X =  2261.501  mm,	Y =    37.528  mm,	Z =    -6.118  mm,
	W =    44.920 deg,	P =     3.025 deg,	R =    -3.029 deg
   GP2:
	UF : 1, UT : 1,
	J1=    90.000 deg,	J2=    90.000 deg
};
P[311]{
   GP1:
	UF : 1, UT : 1,		CONFIG : 'N U T, 0, 0, 0',
	X =  2155.641  mm,	Y =    39.627  mm,	Z =   -15.239  mm,
	W =    44.920 deg,	P =     3.025 deg,	R =    -3.029 deg
   GP2:
	UF : 1, UT : 1,
	J1=    90.000 deg,	J2=    90.000 deg
};
P[312]{
   GP1:
	UF : 1, UT : 1,		CONFIG : 'N U T, 0, 0, 0',
	X =  2213.357  mm,	Y =    37.987  mm,	Z =   -14.278  mm,
	W =    44.920 deg,	P =     3.025 deg,	R =    -3.029 deg
   GP2:
	UF : 1, UT : 1,
	J1=    90.000 deg,	J2=    90.000 deg
};
P[313]{
   GP1:
	UF : 1, UT : 1,		CONFIG : 'N U T, 0, 0, 0',
	X =  2214.573  mm,	Y =    36.787  mm,	Z =   -11.639  mm,
	W =    44.920 deg,	P =     3.025 deg,	R =   -14.180 deg
   GP2:
	UF : 1, UT : 1,
	J1=    90.000 deg,	J2=    90.000 deg
};
P[314]{
   GP1:
	UF : 1, UT : 1,		CONFIG : 'N U T, 0, 0, 0',
	X =  2115.497  mm,	Y =    36.666  mm,	Z =   -20.463  mm,
	W =    44.934 deg,	P =     3.042 deg,	R =     5.570 deg
   GP2:
	UF : 1, UT : 1,
	J1=    90.000 deg,	J2=    90.000 deg
};
P[315]{
   GP1:
	UF : 1, UT : 1,		CONFIG : 'N U T, 0, 0, 0',
	X =  2025.978  mm,	Y =    40.194  mm,	Z =   -20.755  mm,
	W =    44.928 deg,	P =     3.034 deg,	R =     5.584 deg
   GP2:
	UF : 1, UT : 1,
	J1=    90.000 deg,	J2=    90.000 deg
};
P[316]{
   GP1:
	UF : 1, UT : 1,		CONFIG : 'N U T, 0, 0, 0',
	X =  2016.978  mm,	Y =    40.597  mm,	Z =   -22.240  mm,
	W =    44.927 deg,	P =     3.029 deg,	R =    34.553 deg
   GP2:
	UF : 1, UT : 1,
	J1=    90.000 deg,	J2=    90.000 deg
};
P[317]{
   GP1:
	UF : 1, UT : 1,		CONFIG : 'N U T, 0, 0, 0',
	X =  1799.412  mm,	Y =    41.133  mm,	Z =    49.790  mm,
	W =    50.318 deg,	P =     2.533 deg,	R =    12.052 deg
   GP2:
	UF : 1, UT : 1,
	J1=    90.000 deg,	J2=    90.000 deg
};
P[318]{
   GP1:
	UF : 1, UT : 1,		CONFIG : 'N U T, 0, 0, 0',
	X =  1689.959  mm,	Y =    40.113  mm,	Z =    51.381  mm,
	W =    50.325 deg,	P =     2.535 deg,	R =    12.049 deg
   GP2:
	UF : 1, UT : 1,
	J1=    90.000 deg,	J2=    90.000 deg
};
P[319]{
   GP1:
	UF : 1, UT : 1,		CONFIG : 'N U T, 0, 0, 0',
	X =  1672.091  mm,	Y =    39.397  mm,	Z =    51.498  mm,
	W =    55.797 deg,	P =      .895 deg,	R =    26.094 deg
   GP2:
	UF : 1, UT : 1,
	J1=    90.000 deg,	J2=    90.000 deg
};
P[320]{
   GP1:
	UF : 1, UT : 1,		CONFIG : 'N U T, 0, 0, 0',
	X =  1821.553  mm,	Y =    44.041  mm,	Z =    47.838  mm,
	W =    52.757 deg,	P =    -4.415 deg,	R =     3.518 deg
   GP2:
	UF : 1, UT : 1,
	J1=    90.000 deg,	J2=    90.000 deg
};
P[321]{
   GP1:
	UF : 1, UT : 1,		CONFIG : 'N U T, 0, 0, 0',
	X =  1385.322  mm,	Y =    99.987  mm,	Z =    81.524  mm,
	W =   -41.156 deg,	P =    19.919 deg,	R =    36.091 deg
   GP2:
	UF : 1, UT : 1,
	J1=    90.000 deg,	J2=    90.000 deg
};
P[322]{
   GP1:
	UF : 1, UT : 1,		CONFIG : 'N U T, 0, 0, 0',
	X =  1287.575  mm,	Y =   726.729  mm,	Z =   436.468  mm,
	W =   -45.215 deg,	P =    11.103 deg,	R =    59.860 deg
   GP2:
	UF : 1, UT : 1,
	J1=    90.000 deg,	J2=    90.000 deg
};
P[323]{
   GP1:
	UF : 1, UT : 1,		CONFIG : 'N U T, 0, 0, 0',
	X =  2772.800  mm,	Y =  1353.842  mm,	Z =    52.554  mm,
	W =      .247 deg,	P =     2.267 deg,	R =    25.456 deg
   GP2:
	UF : 1, UT : 1,
	J1=    90.000 deg,	J2=    90.000 deg
};
P[324]{
   GP1:
	UF : 1, UT : 1,		CONFIG : 'N U T, 0, 0, 0',
	X =  2849.615  mm,	Y =  1373.219  mm,	Z =     2.246  mm,
	W =      .303 deg,	P =     1.056 deg,	R =    25.442 deg
   GP2:
	UF : 1, UT : 1,
	J1=    89.998 deg,	J2=    90.000 deg
};
P[325]{
   GP1:
	UF : 1, UT : 1,		CONFIG : 'N U B, 0, 0, 0',
	X =   356.032  mm,	Y =    -2.146  mm,	Z =  2424.049  mm,
	W =      .001 deg,	P =   -40.002 deg,	R =     -.005 deg
   GP2:
	UF : 1, UT : 1,
	J1=   -90.000 deg,	J2=    90.000 deg
};
P[326]{
   GP1:
	UF : 1, UT : 1,		CONFIG : 'N U T, 0, 0, 0',
	X =  1109.146  mm,	Y =  -695.879  mm,	Z =  1059.006  mm,
	W =   -45.665 deg,	P =    -3.656 deg,	R =    28.137 deg
   GP2:
	UF : 1, UT : 1,
	J1=   -90.000 deg,	J2=    90.000 deg
};
P[327]{
   GP1:
	UF : 1, UT : 1,		CONFIG : 'N U T, 0, 0, 0',
	X =  2182.795  mm,	Y =   -54.409  mm,	Z =  -297.620  mm,
	W =    -4.848 deg,	P =     4.640 deg,	R =    10.727 deg
   GP2:
	UF : 1, UT : 1,
	J1=    45.000 deg,	J2=   182.246 deg
};
P[328]{
   GP1:
	UF : 1, UT : 1,		CONFIG : 'N U T, 0, 0, 0',
	X =  2785.854  mm,	Y =  1360.233  mm,	Z =    51.016  mm,
	W =      .260 deg,	P =     1.052 deg,	R =    25.457 deg
   GP2:
	UF : 1, UT : 1,
	J1=    90.000 deg,	J2=    90.000 deg
};
P[329]{
   GP1:
	UF : 1, UT : 1,		CONFIG : 'N U T, 0, 0, 0',
	X =  1254.943  mm,	Y =   301.685  mm,	Z =   234.946  mm,
	W =   -61.903 deg,	P =    47.077 deg,	R =    68.180 deg
   GP2:
	UF : 1, UT : 1,
	J1=    90.000 deg,	J2=    90.000 deg
};
P[330]{
   GP1:
	UF : 1, UT : 1,		CONFIG : 'N U T, 0, 0, 0',
	X =  1969.022  mm,	Y =    41.636  mm,	Z =    48.426  mm,
	W =    53.726 deg,	P =    -4.474 deg,	R =     3.443 deg
   GP2:
	UF : 1, UT : 1,
	J1=    90.000 deg,	J2=    90.000 deg
};
P[331]{
   GP1:
	UF : 1, UT : 1,		CONFIG : 'N U T, 0, 0, 0',
	X =  1217.104  mm,	Y =  -169.780  mm,	Z =   187.729  mm,
	W =   -34.745 deg,	P =    30.619 deg,	R =   119.475 deg
   GP2:
	UF : 1, UT : 1,
	J1=    90.000 deg,	J2=    90.000 deg
};
P[332]{
   GP1:
	UF : 1, UT : 1,		CONFIG : 'N U T, 0, 0, 0',
	X =  1573.104  mm,	Y =  -218.075  mm,	Z =    59.729  mm,
	W =   -34.744 deg,	P =    30.618 deg,	R =   128.397 deg
   GP2:
	UF : 1, UT : 1,
	J1=    90.000 deg,	J2=    90.000 deg
};
P[333]{
   GP1:
	UF : 1, UT : 1,		CONFIG : 'N U T, 0, 0, 0',
	X =  1991.252  mm,	Y =    40.726  mm,	Z =    49.738  mm,
	W =    52.869 deg,	P =   -12.269 deg,	R =   -23.050 deg
   GP2:
	UF : 1, UT : 1,
	J1=    90.000 deg,	J2=    90.000 deg
};
P[334]{
   GP1:
	UF : 1, UT : 1,		CONFIG : 'N U T, 0, 0, 0',
	X =  2230.442  mm,	Y =    51.853  mm,	Z =    -5.922  mm,
	W =   -44.607 deg,	P =    -6.682 deg,	R =    -6.729 deg
   GP2:
	UF : 1, UT : 1,
	J1=    90.000 deg,	J2=    90.000 deg
};
P[335]{
   GP1:
	UF : 1, UT : 1,		CONFIG : 'N U T, 0, 0, 1',
	X =  1459.008  mm,	Y =   -74.800  mm,	Z =   199.820  mm,
	W =   -34.742 deg,	P =    30.617 deg,	R =   153.799 deg
   GP2:
	UF : 1, UT : 1,
	J1=    90.000 deg,	J2=    90.000 deg
};
P[336]{
   GP1:
	UF : 1, UT : 1,		CONFIG : 'N U T, 0, 0, 0',
	X =  1319.009  mm,	Y =  -291.799  mm,	Z =   199.820  mm,
	W =    44.863 deg,	P =    -3.871 deg,	R =     -.364 deg
   GP2:
	UF : 1, UT : 1,
	J1=    90.000 deg,	J2=    90.000 deg
};
P[337]{
   GP1:
	UF : 1, UT : 1,		CONFIG : 'N U T, 0, 0, 0',
	X =  2390.009  mm,	Y =  -240.799  mm,	Z =    52.820  mm,
	W =    42.099 deg,	P =    -2.376 deg,	R =   -15.667 deg
   GP2:
	UF : 1, UT : 1,
	J1=    90.000 deg,	J2=    90.000 deg
};
P[338]{
   GP1:
	UF : 1, UT : 1,		CONFIG : 'N U T, 0, 0, 0',
	X =  2264.485  mm,	Y =    52.336  mm,	Z =    -5.439  mm,
	W =   -44.607 deg,	P =    -6.682 deg,	R =    -6.729 deg
   GP2:
	UF : 1, UT : 1,
	J1=    90.000 deg,	J2=    90.000 deg
};
P[339]{
   GP1:
	UF : 1, UT : 1,		CONFIG : 'N U T, 0, 0, 0',
	X =  2141.462  mm,	Y =    52.670  mm,	Z =   -13.878  mm,
	W =   -44.606 deg,	P =    -6.681 deg,	R =    -6.729 deg
   GP2:
	UF : 1, UT : 1,
	J1=    90.000 deg,	J2=    90.000 deg
};
P[340]{
   GP1:
	UF : 1, UT : 1,		CONFIG : 'N U T, 0, 0, 0',
	X =  2502.492  mm,	Y =  -211.230  mm,	Z =    67.973  mm,
	W =    44.580 deg,	P =     6.891 deg,	R =   -21.154 deg
   GP2:
	UF : 1, UT : 1,
	J1=    90.000 deg,	J2=    90.000 deg
};
P[341]{
   GP1:
	UF : 1, UT : 1,		CONFIG : 'N U T, 0, 0, 0',
	X =  2329.524  mm,	Y =  -211.230  mm,	Z =    67.973  mm,
	W =    44.580 deg,	P =     6.891 deg,	R =   -21.154 deg
   GP2:
	UF : 1, UT : 1,
	J1=    90.000 deg,	J2=    90.000 deg
};
P[342]{
   GP1:
	UF : 1, UT : 1,		CONFIG : 'N U T, 0, 0, 0',
	X =  2329.524  mm,	Y =  -124.230  mm,	Z =    67.973  mm,
	W =    44.580 deg,	P =     6.891 deg,	R =   -21.154 deg
   GP2:
	UF : 1, UT : 1,
	J1=    90.000 deg,	J2=    90.000 deg
};
P[343]{
   GP1:
	UF : 1, UT : 1,		CONFIG : 'N U T, 0, 0, 0',
	X =  2208.711  mm,	Y =    51.845  mm,	Z =   -13.000  mm,
	W =   -44.606 deg,	P =    -6.681 deg,	R =    -6.730 deg
   GP2:
	UF : 1, UT : 1,
	J1=    90.000 deg,	J2=    90.000 deg
};
P[344]{
   GP1:
	UF : 1, UT : 1,		CONFIG : 'N U T, 0, 0, 0',
	X =  2214.514  mm,	Y =    56.035  mm,	Z =   -11.445  mm,
	W =   -44.606 deg,	P =    -6.681 deg,	R =     6.841 deg
   GP2:
	UF : 1, UT : 1,
	J1=    90.000 deg,	J2=    90.000 deg
};
P[345]{
   GP1:
	UF : 1, UT : 1,		CONFIG : 'N U T, 0, 0, 0',
	X =  1992.263  mm,	Y =    56.122  mm,	Z =   -19.968  mm,
	W =   -44.607 deg,	P =    -6.682 deg,	R =    -3.024 deg
   GP2:
	UF : 1, UT : 1,
	J1=    90.000 deg,	J2=    90.000 deg
};
P[346]{
   GP1:
	UF : 1, UT : 1,		CONFIG : 'N U T, 0, 0, 0',
	X =  2329.524  mm,	Y =  -124.230  mm,	Z =    67.973  mm,
	W =    44.580 deg,	P =     6.891 deg,	R =   -21.154 deg
   GP2:
	UF : 1, UT : 1,
	J1=    90.000 deg,	J2=    90.000 deg
};
P[347]{
   GP1:
	UF : 1, UT : 1,		CONFIG : 'N U T, 0, 0, 0',
	X =  1069.524  mm,	Y =  -124.230  mm,	Z =   124.973  mm,
	W =    53.137 deg,	P =    27.952 deg,	R =    15.270 deg
   GP2:
	UF : 1, UT : 1,
	J1=    90.000 deg,	J2=    90.000 deg
};
P[348]{
   GP1:
	UF : 1, UT : 1,		CONFIG : 'N U T, 0, 0, 0',
	X =  1062.033  mm,	Y =   -72.059  mm,	Z =  1104.020  mm,
	W =     1.209 deg,	P =    20.107 deg,	R =    63.832 deg
   GP2:
	UF : 1, UT : 1,
	J1=    90.000 deg,	J2=    90.000 deg
};
P[349]{
   GP1:
	UF : 1, UT : 1,		CONFIG : 'N U T, 0, 0, 0',
	X =  1214.600  mm,	Y =   479.028  mm,	Z =   916.465  mm,
	W =    39.867 deg,	P =   -22.888 deg,	R =   -38.695 deg
   GP2:
	UF : 1, UT : 1,
	J1=   -90.000 deg,	J2=   -90.000 deg
};
P[350]{
   GP1:
	UF : 1, UT : 1,		CONFIG : 'N U T, 0, 0, 0',
	X =   713.970  mm,	Y =   812.888  mm,	Z =  1598.123  mm,
	W =    60.754 deg,	P =   -26.996 deg,	R =   -17.604 deg
   GP2:
	UF : 1, UT : 1,
	J1=   -90.000 deg,	J2=   -90.000 deg
};
P[351]{
   GP1:
	UF : 1, UT : 1,		CONFIG : 'N U T, 0, 0, 0',
	X =  1615.600  mm,	Y =   479.028  mm,	Z =   916.465  mm,
	W =    39.867 deg,	P =   -22.888 deg,	R =   -65.014 deg
   GP2:
	UF : 1, UT : 1,
	J1=   -90.000 deg,	J2=   -90.000 deg
};
P[352]{
   GP1:
	UF : 1, UT : 1,		CONFIG : 'N U T, 0, 0, 0',
	X =  2107.423  mm,	Y =    54.740  mm,	Z =   -20.388  mm,
	W =   -44.607 deg,	P =    -6.682 deg,	R =    -3.024 deg
   GP2:
	UF : 1, UT : 1,
	J1=    90.000 deg,	J2=    90.000 deg
};
P[353]{
   GP1:
	UF : 1, UT : 1,		CONFIG : 'N U T, 0, 0, 0',
	X =  2111.262  mm,	Y =    57.036  mm,	Z =   -16.902  mm,
	W =   -42.118 deg,	P =   -17.568 deg,	R =    21.832 deg
   GP2:
	UF : 1, UT : 1,
	J1=    90.000 deg,	J2=    90.000 deg
};
P[354]{
   GP1:
	UF : 1, UT : 1,		CONFIG : 'N U T, 0, 0, 0',
	X =  2012.717  mm,	Y =    84.636  mm,	Z =    -8.736  mm,
	W =   -45.251 deg,	P =    -8.450 deg,	R =  -108.138 deg
   GP2:
	UF : 1, UT : 1,
	J1=    90.000 deg,	J2=   100.000 deg
};
P[355]{
   GP1:
	UF : 1, UT : 1,		CONFIG : 'N U T, 0, 0, 0',
	X =  2008.359  mm,	Y =  -137.141  mm,	Z =   -45.703  mm,
	W =   -45.251 deg,	P =    -8.450 deg,	R =   -86.328 deg
   GP2:
	UF : 1, UT : 1,
	J1=    90.000 deg,	J2=   100.000 deg
};
P[356]{
   GP1:
	UF : 1, UT : 1,		CONFIG : 'N U T, 0, 0, 0',
	X =  2753.412  mm,	Y =   160.459  mm,	Z =   180.671  mm,
	W =     2.791 deg,	P =    -7.674 deg,	R =   -18.462 deg
   GP2:
	UF : 1, UT : 1,
	J1=    90.000 deg,	J2=   135.000 deg
};
P[357]{
   GP1:
	UF : 1, UT : 1,		CONFIG : 'N U T, 0, 0, 0',
	X =  2867.805  mm,	Y =   160.634  mm,	Z =   182.471  mm,
	W =     9.502 deg,	P =   -26.582 deg,	R =   -20.495 deg
   GP2:
	UF : 1, UT : 1,
	J1=    89.999 deg,	J2=   135.000 deg
};
P[358]{
   GP1:
	UF : 1, UT : 1,		CONFIG : 'N U T, 0, 0, 0',
	X =  2378.956  mm,	Y =   265.120  mm,	Z =    86.366  mm,
	W =     1.850 deg,	P =     -.182 deg,	R =      .942 deg
   GP2:
	UF : 1, UT : 1,
	J1=    90.000 deg,	J2=   135.000 deg
};
P[359]{
   GP1:
	UF : 1, UT : 1,		CONFIG : 'N U T, 0, 0, 0',
	X =  2754.391  mm,	Y =   263.612  mm,	Z =    86.366  mm,
	W =     1.733 deg,	P =    -7.250 deg,	R =      .949 deg
   GP2:
	UF : 1, UT : 1,
	J1=    90.000 deg,	J2=   135.000 deg
};
P[360]{
   GP1:
	UF : 1, UT : 1,		CONFIG : 'N U T, 0, 0, 0',
	X =  1704.637  mm,	Y =   898.337  mm,	Z =  1001.782  mm,
	W =   -20.210 deg,	P =   -41.106 deg,	R =     1.246 deg
   GP2:
	UF : 1, UT : 1,
	J1=   -90.000 deg,	J2=   -90.000 deg
};
P[361]{
   GP1:
	UF : 1, UT : 1,		CONFIG : 'N U T, 0, 0, 0',
	X =  1682.137  mm,	Y =   345.195  mm,	Z =   941.171  mm,
	W =    42.022 deg,	P =   -15.891 deg,	R =   -33.571 deg
   GP2:
	UF : 1, UT : 1,
	J1=   -90.000 deg,	J2=   -90.000 deg
};
P[362]{
   GP1:
	UF : 1, UT : 1,		CONFIG : 'N U T, 0, 0, 0',
	X =  2068.312  mm,	Y =   107.394  mm,	Z =   -18.582  mm,
	W =    37.933 deg,	P =    17.387 deg,	R =   -97.672 deg
   GP2:
	UF : 1, UT : 1,
	J1=    90.000 deg,	J2=    90.000 deg
};
P[363]{
   GP1:
	UF : 1, UT : 1,		CONFIG : 'N U T, 0, 0, 0',
	X =  2109.723  mm,	Y =    72.505  mm,	Z =   -21.222  mm,
	W =    37.933 deg,	P =    17.387 deg,	R =  -104.287 deg
   GP2:
	UF : 1, UT : 1,
	J1=    90.000 deg,	J2=    90.000 deg
};
P[364]{
   GP1:
	UF : 1, UT : 1,		CONFIG : 'N U T, 0, 0, -1',
	X =  2115.592  mm,	Y =    62.473  mm,	Z =   -16.026  mm,
	W =    44.181 deg,	P =    21.261 deg,	R =  -126.963 deg
   GP2:
	UF : 1, UT : 1,
	J1=    90.000 deg,	J2=    90.000 deg
};
P[365]{
   GP1:
	UF : 1, UT : 1,		CONFIG : 'N U T, 0, 0, 0',
	X =  2357.041  mm,	Y =   -23.041  mm,	Z =    82.290  mm,
	W =   -26.718 deg,	P =   -22.770 deg,	R =   -10.639 deg
   GP2:
	UF : 1, UT : 1,
	J1=    90.000 deg,	J2=   100.000 deg
};
P[366]{
   GP1:
	UF : 1, UT : 1,		CONFIG : 'N U T, 0, 0, 0',
	X =  1685.743  mm,	Y =    59.810  mm,	Z =   -17.917  mm,
	W =   -42.807 deg,	P =    15.441 deg,	R =    16.037 deg
   GP2:
	UF : 1, UT : 1,
	J1=    90.000 deg,	J2=    90.000 deg
};
P[367]{
   GP1:
	UF : 1, UT : 1,		CONFIG : 'N U T, 0, 0, 0',
	X =  1855.998  mm,	Y =   173.909  mm,	Z =   960.367  mm,
	W =    58.350 deg,	P =   -26.173 deg,	R =   -73.280 deg
   GP2:
	UF : 1, UT : 1,
	J1=   -90.000 deg,	J2=   -90.000 deg
};
P[368]{
   GP1:
	UF : 1, UT : 1,		CONFIG : 'N U T, 0, 0, 0',
	X =  1291.698  mm,	Y =   195.066  mm,	Z =   960.367  mm,
	W =    58.350 deg,	P =   -26.173 deg,	R =   -73.280 deg
   GP2:
	UF : 1, UT : 1,
	J1=   -90.000 deg,	J2=   -90.000 deg
};
P[369]{
   GP1:
	UF : 1, UT : 1,		CONFIG : 'N U T, 0, 0, 0',
	X =  1652.429  mm,	Y =    58.946  mm,	Z =   -19.364  mm,
	W =   -42.810 deg,	P =    15.442 deg,	R =    16.034 deg
   GP2:
	UF : 1, UT : 1,
	J1=    90.000 deg,	J2=    90.000 deg
};
P[370]{
   GP1:
	UF : 1, UT : 1,		CONFIG : 'N U T, 0, 0, 0',
	X =  1640.987  mm,	Y =    56.683  mm,	Z =   -21.519  mm,
	W =   -42.181 deg,	P =    15.522 deg,	R =    -8.109 deg
   GP2:
	UF : 1, UT : 1,
	J1=    90.000 deg,	J2=    90.000 deg
};
P[371]{
   GP1:
	UF : 1, UT : 1,		CONFIG : 'N U T, 0, 0, 0',
	X =  1433.073  mm,	Y =  -528.643  mm,	Z =   576.275  mm,
	W =    -5.611 deg,	P =   -10.020 deg,	R =     8.093 deg
   GP2:
	UF : 1, UT : 1,
	J1=    90.000 deg,	J2=  -100.000 deg
};
P[372]{
   GP1:
	UF : 1, UT : 1,		CONFIG : 'N U T, 0, 0, 0',
	X =  1558.148  mm,	Y =   135.723  mm,	Z =   206.394  mm,
	W =   -46.360 deg,	P =    11.199 deg,	R =    10.858 deg
   GP2:
	UF : 1, UT : 1,
	J1=    90.000 deg,	J2=   -90.000 deg
};
P[373]{
   GP1:
	UF : 1, UT : 1,		CONFIG : 'N U T, 0, 0, 0',
	X =  2022.992  mm,	Y =   -45.728  mm,	Z =     2.837  mm,
	W =   -43.918 deg,	P =    -5.993 deg,	R =   -30.730 deg
   GP2:
	UF : 1, UT : 1,
	J1=    90.000 deg,	J2=   -90.000 deg
};
P[374]{
   GP1:
	UF : 1, UT : 1,		CONFIG : 'N U T, 0, 0, 0',
	X =  1637.701  mm,	Y =    59.485  mm,	Z =   -19.665  mm,
	W =   -38.593 deg,	P =    25.218 deg,	R =   -16.905 deg
   GP2:
	UF : 1, UT : 1,
	J1=    90.000 deg,	J2=    90.000 deg
};
P[375]{
   GP1:
	UF : 1, UT : 1,		CONFIG : 'N U T, 0, 0, 0',
	X =  1608.736  mm,	Y =    83.348  mm,	Z =   -24.399  mm,
	W =   -38.593 deg,	P =    25.219 deg,	R =   -16.905 deg
   GP2:
	UF : 1, UT : 1,
	J1=    90.000 deg,	J2=    90.000 deg
};
P[376]{
   GP1:
	UF : 1, UT : 1,		CONFIG : 'N U T, 0, 0, 0',
	X =  2053.353  mm,	Y =   209.744  mm,	Z =   328.977  mm,
	W =   -44.718 deg,	P =   -17.447 deg,	R =    -6.431 deg
   GP2:
	UF : 1, UT : 1,
	J1=    90.000 deg,	J2=   100.000 deg
};
P[377]{
   GP1:
	UF : 1, UT : 1,		CONFIG : 'N U T, 0, 0, 0',
	X =  1074.532  mm,	Y =  -506.968  mm,	Z =  1238.459  mm,
	W =     -.673 deg,	P =   -46.105 deg,	R =     9.949 deg
   GP2:
	UF : 1, UT : 1,
	J1=   -90.000 deg,	J2=    90.000 deg
};
P[378]{
   GP1:
	UF : 1, UT : 1,		CONFIG : 'N U T, 0, 0, 0',
	X =  1359.532  mm,	Y =  -506.968  mm,	Z =   962.459  mm,
	W =     -.673 deg,	P =   -46.105 deg,	R =     9.949 deg
   GP2:
	UF : 1, UT : 1,
	J1=   -90.000 deg,	J2=    90.000 deg
};
P[379]{
   GP1:
	UF : 1, UT : 1,		CONFIG : 'N U T, 0, 0, 0',
	X =  1645.943  mm,	Y =  -472.973  mm,	Z =   885.320  mm,
	W =   -29.059 deg,	P =   -38.116 deg,	R =    41.980 deg
   GP2:
	UF : 1, UT : 1,
	J1=   -90.000 deg,	J2=    90.000 deg
};
P[380]{
   GP1:
	UF : 1, UT : 1,		CONFIG : 'N U T, 0, 0, 0',
	X =  1214.623  mm,	Y =   483.357  mm,	Z =   914.016  mm,
	W =   -25.369 deg,	P =    11.963 deg,	R =   -19.314 deg
   GP2:
	UF : 1, UT : 1,
	J1=    90.000 deg,	J2=   100.000 deg
};
P[381]{
   GP1:
	UF : 1, UT : 1,		CONFIG : 'N U T, 0, 0, -1',
	X =  1626.194  mm,	Y =   455.887  mm,	Z =  1153.200  mm,
	W =     5.544 deg,	P =    60.170 deg,	R =  -166.026 deg
   GP2:
	UF : 1, UT : 1,
	J1=    90.000 deg,	J2=    90.000 deg
};
P[382]{
   GP1:
	UF : 1, UT : 1,		CONFIG : 'N U T, 0, 0, 0',
	X =  1585.662  mm,	Y =   101.135  mm,	Z =   -21.859  mm,
	W =   -45.000 deg,	P =    -3.170 deg,	R =      .426 deg
   GP2:
	UF : 1, UT : 1,
	J1=    90.000 deg,	J2=    90.000 deg
};
P[383]{
   GP1:
	UF : 1, UT : 1,		CONFIG : 'N U T, 0, 0, 0',
	X =  1556.810  mm,	Y =    69.060  mm,	Z =   -21.622  mm,
	W =   -45.449 deg,	P =    19.944 deg,	R =    98.982 deg
   GP2:
	UF : 1, UT : 1,
	J1=    90.000 deg,	J2=    90.000 deg
};
P[384]{
   GP1:
	UF : 1, UT : 1,		CONFIG : 'N U T, 0, 0, 0',
	X =  1551.240  mm,	Y =    28.811  mm,	Z =   -19.922  mm,
	W =   -45.337 deg,	P =    20.062 deg,	R =    97.887 deg
   GP2:
	UF : 1, UT : 1,
	J1=    90.000 deg,	J2=    90.000 deg
};
P[385]{
   GP1:
	UF : 1, UT : 1,		CONFIG : 'N U T, 0, 0, 0',
	X =  1551.443  mm,	Y =    22.198  mm,	Z =   -20.367  mm,
	W =   -45.343 deg,	P =    20.068 deg,	R =    97.646 deg
   GP2:
	UF : 1, UT : 1,
	J1=    90.000 deg,	J2=    90.000 deg
};
P[386]{
   GP1:
	UF : 1, UT : 1,		CONFIG : 'N U T, 0, 0, 0',
	X =  1549.407  mm,	Y =    21.768  mm,	Z =   -17.950  mm,
	W =   -41.210 deg,	P =    19.947 deg,	R =    34.862 deg
   GP2:
	UF : 1, UT : 1,
	J1=    90.000 deg,	J2=    90.000 deg
};
P[387]{
   GP1:
	UF : 1, UT : 1,		CONFIG : 'N U T, 0, 0, 0',
	X =  1540.684  mm,	Y =    20.490  mm,	Z =   -17.846  mm,
	W =   -41.215 deg,	P =    19.945 deg,	R =    34.866 deg
   GP2:
	UF : 1, UT : 1,
	J1=    90.000 deg,	J2=    90.000 deg
};
P[388]{
   GP1:
	UF : 1, UT : 1,		CONFIG : 'N U T, 0, 0, 0',
	X =  1597.869  mm,	Y =  -854.871  mm,	Z =   914.402  mm,
	W =   -20.245 deg,	P =   -41.090 deg,	R =    57.299 deg
   GP2:
	UF : 1, UT : 1,
	J1=   -90.000 deg,	J2=    90.000 deg
};
P[389]{
   GP1:
	UF : 1, UT : 1,		CONFIG : 'N U T, 0, 0, 0',
	X =  1597.869  mm,	Y =  -357.729  mm,	Z =   914.402  mm,
	W =   -53.336 deg,	P =     2.108 deg,	R =    49.603 deg
   GP2:
	UF : 1, UT : 1,
	J1=   -90.000 deg,	J2=    90.000 deg
};
P[390]{
   GP1:
	UF : 1, UT : 1,		CONFIG : 'N U T, 0, 0, 0',
	X =  2866.453  mm,	Y =  1420.346  mm,	Z =   -11.619  mm,
	W =     -.178 deg,	P =    -1.186 deg,	R =    26.508 deg
   GP2:
	UF : 1, UT : 1,
	J1=    90.000 deg,	J2=    90.000 deg
};
P[391]{
   GP1:
	UF : 1, UT : 1,		CONFIG : 'N U T, 0, 0, 0',
	X =  2866.454  mm,	Y =  1403.775  mm,	Z =   -11.619  mm,
	W =     -.178 deg,	P =    -1.186 deg,	R =    26.508 deg
   GP2:
	UF : 1, UT : 1,
	J1=    90.000 deg,	J2=    90.000 deg
};
P[395]{
   GP1:
	UF : 1, UT : 1,		CONFIG : 'N U T, 0, 0, 0',
	X =  1813.190  mm,	Y =  -222.628  mm,	Z =   892.611  mm,
	W =   -54.261 deg,	P =    -6.374 deg,	R =    77.692 deg
   GP2:
	UF : 1, UT : 1,
	J1=   -90.000 deg,	J2=    90.000 deg
};
P[396]{
   GP1:
	UF : 1, UT : 1,		CONFIG : 'N U T, 0, 0, 0',
	X =  1480.982  mm,	Y =  -280.121  mm,	Z =   888.392  mm,
	W =   -52.435 deg,	P =    -5.968 deg,	R =    77.563 deg
   GP2:
	UF : 1, UT : 1,
	J1=   -90.000 deg,	J2=    90.000 deg
};
P[397]{
   GP1:
	UF : 1, UT : 1,		CONFIG : 'N U T, 0, 0, -1',
	X =  2103.205  mm,	Y =   181.792  mm,	Z =  1015.411  mm,
	W =     -.647 deg,	P =    55.219 deg,	R =   156.602 deg
   GP2:
	UF : 1, UT : 1,
	J1=    90.000 deg,	J2=    90.000 deg
};
P[399]{
   GP1:
	UF : 1, UT : 1,		CONFIG : 'N U T, 0, 0, 1',
	X =  1651.536  mm,	Y =  -219.100  mm,	Z =   -19.888  mm,
	W =   -32.939 deg,	P =    29.350 deg,	R =   129.300 deg
   GP2:
	UF : 1, UT : 1,
	J1=    90.000 deg,	J2=    90.000 deg
};
P[400]{
   GP1:
	UF : 1, UT : 1,		CONFIG : 'N U T, 0, 0, 1',
	X =  1652.465  mm,	Y =    20.682  mm,	Z =   -20.854  mm,
	W =   -34.233 deg,	P =    30.069 deg,	R =   141.356 deg
   GP2:
	UF : 1, UT : 1,
	J1=    90.000 deg,	J2=    90.000 deg
};
P[401]{
   GP1:
	UF : 1, UT : 1,		CONFIG : 'N U T, 0, 0, 0',
	X =  2351.061  mm,	Y =  -179.371  mm,	Z =   -13.077  mm,
	W =    44.587 deg,	P =     6.899 deg,	R =    -6.951 deg
   GP2:
	UF : 1, UT : 1,
	J1=    90.000 deg,	J2=    90.000 deg
};
P[402]{
   GP1:
	UF : 1, UT : 1,		CONFIG : 'N U T, 0, 0, 0',
	X =  2518.615  mm,	Y =  -178.195  mm,	Z =   -13.758  mm,
	W =    44.582 deg,	P =     6.892 deg,	R =    -6.941 deg
   GP2:
	UF : 1, UT : 1,
	J1=    90.000 deg,	J2=    90.000 deg
};
P[403]{
   GP1:
	UF : 1, UT : 1,		CONFIG : 'N U T, 0, 0, 0',
	X =  2352.052  mm,	Y =   -90.042  mm,	Z =   -15.707  mm,
	W =    43.242 deg,	P =    13.891 deg,	R =   -18.605 deg
   GP2:
	UF : 1, UT : 1,
	J1=    90.000 deg,	J2=    90.000 deg
};
P[404]{
   GP1:
	UF : 1, UT : 1,		CONFIG : 'N U T, 0, 0, 0',
	X =  2404.409  mm,	Y =   -89.953  mm,	Z =   -14.975  mm,
	W =    43.244 deg,	P =    13.890 deg,	R =   -18.607 deg
   GP2:
	UF : 1, UT : 1,
	J1=    90.000 deg,	J2=    90.000 deg
};
P[405]{
   GP1:
	UF : 1, UT : 1,		CONFIG : 'N U T, 0, 0, 0',
	X =  2423.248  mm,	Y =   -92.540  mm,	Z =    -8.646  mm,
	W =    42.728 deg,	P =    13.810 deg,	R =   -51.889 deg
   GP2:
	UF : 1, UT : 1,
	J1=    89.998 deg,	J2=    90.000 deg
};
P[406]{
   GP1:
	UF : 1, UT : 1,		CONFIG : 'N U T, 0, 0, 0',
	X =  1684.563  mm,	Y =   458.656  mm,	Z =   830.406  mm,
	W =    39.866 deg,	P =   -22.888 deg,	R =   -65.013 deg
   GP2:
	UF : 1, UT : 1,
	J1=   -90.000 deg,	J2=   -90.000 deg
};
P[407]{
   GP1:
	UF : 1, UT : 1,		CONFIG : 'N U T, 0, 0, 0',
	X =  1685.493  mm,	Y =   473.679  mm,	Z =   828.230  mm,
	W =    39.866 deg,	P =   -22.887 deg,	R =   -65.013 deg
   GP2:
	UF : 1, UT : 1,
	J1=   -90.000 deg,	J2=   -90.000 deg
};
P[408]{
   GP1:
	UF : 1, UT : 1,		CONFIG : 'N U T, 0, 0, 0',
	X =  1685.563  mm,	Y =   480.822  mm,	Z =   829.093  mm,
	W =    39.867 deg,	P =   -22.888 deg,	R =   -69.837 deg
   GP2:
	UF : 1, UT : 1,
	J1=   -90.000 deg,	J2=   -90.000 deg
};
P[409]{
   GP1:
	UF : 1, UT : 1,		CONFIG : 'N U T, 0, 0, 0',
	X =  1687.491  mm,	Y =   484.680  mm,	Z =   827.711  mm,
	W =    39.867 deg,	P =   -22.888 deg,	R =   -70.971 deg
   GP2:
	UF : 1, UT : 1,
	J1=   -90.000 deg,	J2=   -90.000 deg
};
P[410]{
   GP1:
	UF : 1, UT : 1,		CONFIG : 'N U T, 0, 0, 0',
	X =  1708.839  mm,	Y =   554.633  mm,	Z =   827.423  mm,
	W =    39.871 deg,	P =   -22.884 deg,	R =   -70.976 deg
   GP2:
	UF : 1, UT : 1,
	J1=   -90.000 deg,	J2=   -90.000 deg
};
P[411]{
   GP1:
	UF : 1, UT : 1,		CONFIG : 'N U T, 0, 0, 0',
	X =  1711.676  mm,	Y =   557.080  mm,	Z =   826.531  mm,
	W =    39.870 deg,	P =   -22.884 deg,	R =   -74.846 deg
   GP2:
	UF : 1, UT : 1,
	J1=   -90.000 deg,	J2=   -90.000 deg
};
P[412]{
   GP1:
	UF : 1, UT : 1,		CONFIG : 'N U T, 0, 0, 0',
	X =  2054.302  mm,	Y =   204.441  mm,	Z =   988.994  mm,
	W =      .815 deg,	P =    36.667 deg,	R =   159.784 deg
   GP2:
	UF : 1, UT : 1,
	J1=    90.000 deg,	J2=    90.000 deg
};
P[413]{
   GP1:
	UF : 1, UT : 1,		CONFIG : 'N U T, 0, 0, 0',
	X =  2128.801  mm,	Y =   250.942  mm,	Z =   983.493  mm,
	W =    -8.588 deg,	P =    43.492 deg,	R =    86.611 deg
   GP2:
	UF : 1, UT : 1,
	J1=    90.000 deg,	J2=    90.000 deg
};
P[414]{
   GP1:
	UF : 1, UT : 1,		CONFIG : 'N U T, 0, 0, 0',
	X =  1712.809  mm,	Y =   560.962  mm,	Z =   826.801  mm,
	W =    39.866 deg,	P =   -22.883 deg,	R =   -82.536 deg
   GP2:
	UF : 1, UT : 1,
	J1=   -90.000 deg,	J2=   -90.000 deg
};
P[415]{
   GP1:
	UF : 1, UT : 1,		CONFIG : 'N U T, 0, 0, 0',
	X =  1845.680  mm,	Y =   825.086  mm,	Z =   832.601  mm,
	W =    14.309 deg,	P =   -43.038 deg,	R =   -40.623 deg
   GP2:
	UF : 1, UT : 1,
	J1=   -89.991 deg,	J2=   -89.999 deg
};
P[416]{
   GP1:
	UF : 1, UT : 1,		CONFIG : 'N U T, 0, 0, 0',
	X =  1698.333  mm,	Y =   426.907  mm,	Z =   830.357  mm,
	W =    43.050 deg,	P =   -14.373 deg,	R =   -45.079 deg
   GP2:
	UF : 1, UT : 1,
	J1=   -90.000 deg,	J2=   -90.000 deg
};
P[417]{
   GP1:
	UF : 1, UT : 1,		CONFIG : 'N U T, 0, 0, 0',
	X =  1839.303  mm,	Y =   266.347  mm,	Z =   829.243  mm,
	W =    43.053 deg,	P =   -14.369 deg,	R =   -45.082 deg
   GP2:
	UF : 1, UT : 1,
	J1=   -90.000 deg,	J2=   -90.000 deg
};
P[418]{
   GP1:
	UF : 1, UT : 1,		CONFIG : 'N U T, 0, 0, 0',
	X =  1847.539  mm,	Y =   258.366  mm,	Z =   830.212  mm,
	W =    43.049 deg,	P =   -14.375 deg,	R =   -42.871 deg
   GP2:
	UF : 1, UT : 1,
	J1=   -90.000 deg,	J2=   -90.000 deg
};
P[419]{
   GP1:
	UF : 1, UT : 1,		CONFIG : 'N U T, 0, 0, 0',
	X =  1859.538  mm,	Y =   247.937  mm,	Z =   830.256  mm,
	W =    43.049 deg,	P =   -14.375 deg,	R =   -40.829 deg
   GP2:
	UF : 1, UT : 1,
	J1=   -90.000 deg,	J2=   -90.000 deg
};
P[420]{
   GP1:
	UF : 1, UT : 1,		CONFIG : 'N U T, 0, 0, 0',
	X =  1923.179  mm,	Y =   200.865  mm,	Z =   829.012  mm,
	W =    43.049 deg,	P =   -14.374 deg,	R =   -40.829 deg
   GP2:
	UF : 1, UT : 1,
	J1=   -90.000 deg,	J2=   -90.000 deg
};
P[421]{
   GP1:
	UF : 1, UT : 1,		CONFIG : 'N U T, 0, 0, 0',
	X =  1678.881  mm,	Y =  -469.975  mm,	Z =   829.150  mm,
	W =   -28.314 deg,	P =   -37.469 deg,	R =    36.647 deg
   GP2:
	UF : 1, UT : 1,
	J1=   -90.000 deg,	J2=    90.000 deg
};
P[422]{
   GP1:
	UF : 1, UT : 1,		CONFIG : 'N U T, 0, 0, 0',
	X =  1682.926  mm,	Y =  -487.189  mm,	Z =   826.659  mm,
	W =   -28.322 deg,	P =   -37.469 deg,	R =    36.650 deg
   GP2:
	UF : 1, UT : 1,
	J1=   -90.000 deg,	J2=    90.000 deg
};
P[423]{
   GP1:
	UF : 1, UT : 1,		CONFIG : 'N U T, 0, 0, 0',
	X =  1682.542  mm,	Y =  -491.734  mm,	Z =   828.424  mm,
	W =   -28.334 deg,	P =   -37.464 deg,	R =    39.731 deg
   GP2:
	UF : 1, UT : 1,
	J1=   -90.000 deg,	J2=    90.000 deg
};
P[424]{
   GP1:
	UF : 1, UT : 1,		CONFIG : 'N U T, 0, 0, 0',
	X =  1683.217  mm,	Y =  -494.546  mm,	Z =   827.297  mm,
	W =   -28.322 deg,	P =   -37.469 deg,	R =    41.171 deg
   GP2:
	UF : 1, UT : 1,
	J1=   -90.000 deg,	J2=    90.000 deg
};
P[425]{
   GP1:
	UF : 1, UT : 1,		CONFIG : 'N U T, 0, 0, 0',
	X =  1707.638  mm,	Y =  -565.332  mm,	Z =   825.835  mm,
	W =   -28.322 deg,	P =   -37.469 deg,	R =    41.171 deg
   GP2:
	UF : 1, UT : 1,
	J1=   -90.000 deg,	J2=    90.000 deg
};
P[426]{
   GP1:
	UF : 1, UT : 1,		CONFIG : 'N U T, 0, 0, 0',
	X =  1709.098  mm,	Y =  -569.548  mm,	Z =   825.685  mm,
	W =   -28.322 deg,	P =   -37.469 deg,	R =    48.505 deg
   GP2:
	UF : 1, UT : 1,
	J1=   -90.000 deg,	J2=    90.000 deg
};
P[427]{
   GP1:
	UF : 1, UT : 1,		CONFIG : 'N U T, 0, 0, 0',
	X =  1713.633  mm,	Y =  -574.840  mm,	Z =   824.222  mm,
	W =   -28.328 deg,	P =   -37.465 deg,	R =    55.403 deg
   GP2:
	UF : 1, UT : 1,
	J1=   -90.000 deg,	J2=    90.000 deg
};
P[428]{
   GP1:
	UF : 1, UT : 1,		CONFIG : 'N U T, 0, 0, 0',
	X =  1842.146  mm,	Y =  -829.157  mm,	Z =   829.639  mm,
	W =   -28.322 deg,	P =   -37.469 deg,	R =    50.636 deg
   GP2:
	UF : 1, UT : 1,
	J1=   -90.000 deg,	J2=    90.000 deg
};
P[429]{
   GP1:
	UF : 1, UT : 1,		CONFIG : 'N U T, 0, 0, 0',
	X =  1690.304  mm,	Y =  -437.670  mm,	Z =   830.884  mm,
	W =   -39.460 deg,	P =    -8.334 deg,	R =    42.657 deg
   GP2:
	UF : 1, UT : 1,
	J1=   -90.000 deg,	J2=    90.000 deg
};
P[430]{
   GP1:
	UF : 1, UT : 1,		CONFIG : 'N U T, 0, 0, 0',
	X =  1836.271  mm,	Y =  -275.564  mm,	Z =   827.815  mm,
	W =   -39.460 deg,	P =    -8.334 deg,	R =    42.657 deg
   GP2:
	UF : 1, UT : 1,
	J1=   -90.000 deg,	J2=    90.000 deg
};
P[431]{
   GP1:
	UF : 1, UT : 1,		CONFIG : 'N U T, 0, 0, 0',
	X =  1848.380  mm,	Y =  -264.272  mm,	Z =   828.029  mm,
	W =   -39.460 deg,	P =    -8.334 deg,	R =    38.620 deg
   GP2:
	UF : 1, UT : 1,
	J1=   -90.000 deg,	J2=    90.000 deg
};
P[432]{
   GP1:
	UF : 1, UT : 1,		CONFIG : 'N U T, 0, 0, 0',
	X =  2643.424  mm,	Y =  -135.910  mm,	Z =   990.550  mm,
	W =   -36.400 deg,	P =    28.534 deg,	R =    31.709 deg
   GP2:
	UF : 1, UT : 1,
	J1=    90.000 deg,	J2=    90.000 deg
};
P[433]{
   GP1:
	UF : 1, UT : 1,		CONFIG : 'N U T, 0, 0, 0',
	X =   983.140  mm,	Y =    19.420  mm,	Z =   990.550  mm,
	W =   -36.400 deg,	P =    28.534 deg,	R =    23.998 deg
   GP2:
	UF : 1, UT : 1,
	J1=    90.000 deg,	J2=    90.000 deg
};
P[434]{
   GP1:
	UF : 1, UT : 1,		CONFIG : 'N U T, 0, 0, 0',
	X =   983.140  mm,	Y =  -212.416  mm,	Z =   990.550  mm,
	W =   -43.636 deg,	P =   -12.296 deg,	R =    70.660 deg
   GP2:
	UF : 1, UT : 1,
	J1=    80.000 deg,	J2=    90.000 deg
};
P[435]{
   GP1:
	UF : 1, UT : 1,		CONFIG : 'N U T, 0, 0, 0',
	X =  1995.140  mm,	Y =  -212.416  mm,	Z =   320.550  mm,
	W =   -43.636 deg,	P =   -12.296 deg,	R =    70.660 deg
   GP2:
	UF : 1, UT : 1,
	J1=    80.000 deg,	J2=    90.000 deg
};
P[436]{
   GP1:
	UF : 1, UT : 1,		CONFIG : 'N U T, 0, 0, 0',
	X =  2018.730  mm,	Y =   -25.769  mm,	Z =   130.343  mm,
	W =   -38.665 deg,	P =    -2.420 deg,	R =   142.728 deg
   GP2:
	UF : 1, UT : 1,
	J1=    80.000 deg,	J2=    90.000 deg
};
P[437]{
   GP1:
	UF : 1, UT : 1,		CONFIG : 'N U T, 0, 0, 0',
	X =  1862.737  mm,	Y =  -253.785  mm,	Z =   829.403  mm,
	W =   -39.460 deg,	P =    -8.334 deg,	R =    41.372 deg
   GP2:
	UF : 1, UT : 1,
	J1=   -90.000 deg,	J2=    90.000 deg
};
P[438]{
   GP1:
	UF : 1, UT : 1,		CONFIG : 'N U T, 0, 0, 0',
	X =  1935.611  mm,	Y =  -199.637  mm,	Z =   827.419  mm,
	W =   -39.460 deg,	P =    -8.334 deg,	R =    45.243 deg
   GP2:
	UF : 1, UT : 1,
	J1=   -90.000 deg,	J2=    90.000 deg
};
P[439]{
   GP1:
	UF : 1, UT : 1,		CONFIG : 'N U T, 0, 0, 0',
	X =  2344.158  mm,	Y =   -61.498  mm,	Z =   837.144  mm,
	W =     4.733 deg,	P =    44.799 deg,	R =    66.706 deg
   GP2:
	UF : 1, UT : 1,
	J1=    90.000 deg,	J2=    90.000 deg
};
P[440]{
   GP1:
	UF : 1, UT : 1,		CONFIG : 'N U T, 0, 0, 0',
	X =  2404.770  mm,	Y =   -93.993  mm,	Z =   837.387  mm,
	W =     4.736 deg,	P =    44.803 deg,	R =    66.702 deg
   GP2:
	UF : 1, UT : 1,
	J1=    90.000 deg,	J2=    90.000 deg
};
P[441]{
   GP1:
	UF : 1, UT : 1,		CONFIG : 'N U T, 0, 0, 0',
	X =  2400.549  mm,	Y =  -120.824  mm,	Z =   838.185  mm,
	W =   -19.419 deg,	P =    41.428 deg,	R =   -56.052 deg
   GP2:
	UF : 1, UT : 1,
	J1=    90.000 deg,	J2=    90.000 deg
};
P[442]{
   GP1:
	UF : 1, UT : 1,		CONFIG : 'N U T, 0, 0, 0',
	X =  2411.665  mm,	Y =  -100.428  mm,	Z =   838.269  mm,
	W =   -19.426 deg,	P =    41.428 deg,	R =   -56.049 deg
   GP2:
	UF : 1, UT : 1,
	J1=    90.000 deg,	J2=    90.000 deg
};
P[443]{
   GP1:
	UF : 1, UT : 1,		CONFIG : 'N U T, 0, 0, 0',
	X =  2329.816  mm,	Y =   -87.227  mm,	Z =   839.756  mm,
	W =    34.022 deg,	P =    31.444 deg,	R =   -66.610 deg
   GP2:
	UF : 1, UT : 1,
	J1=    90.000 deg,	J2=    90.000 deg
};
P[444]{
   GP1:
	UF : 1, UT : 1,		CONFIG : 'N U T, 0, 0, 0',
	X =  2393.327  mm,	Y =  -122.227  mm,	Z =   840.237  mm,
	W =    34.022 deg,	P =    31.444 deg,	R =   -66.610 deg
   GP2:
	UF : 1, UT : 1,
	J1=    90.000 deg,	J2=    90.000 deg
};
P[445]{
   GP1:
	UF : 1, UT : 1,		CONFIG : 'N U T, 0, 0, 0',
	X =  2519.938  mm,	Y =   -81.372  mm,	Z =   -32.158  mm,
	W =   -31.368 deg,	P =   -16.422 deg,	R =   -28.761 deg
   GP2:
	UF : 1, UT : 1,
	J1=    90.000 deg,	J2=   100.000 deg
};
P[446]{
   GP1:
	UF : 1, UT : 1,		CONFIG : 'N U T, 0, 0, 0',
	X =  2482.458  mm,	Y =   -80.069  mm,	Z =   -28.898  mm,
	W =   -25.037 deg,	P =   -25.315 deg,	R =   -46.367 deg
   GP2:
	UF : 1, UT : 1,
	J1=    90.000 deg,	J2=   100.000 deg
};
P[447]{
   GP1:
	UF : 1, UT : 1,		CONFIG : 'N U T, 0, 0, 0',
	X =  2453.629  mm,	Y =   -82.007  mm,	Z =   -26.243  mm,
	W =   -25.039 deg,	P =   -25.325 deg,	R =   -79.891 deg
   GP2:
	UF : 1, UT : 1,
	J1=    90.000 deg,	J2=   100.000 deg
};
P[448]{
   GP1:
	UF : 1, UT : 1,		CONFIG : 'N U T, 0, 0, 0',
	X =  2351.765  mm,	Y =   -85.833  mm,	Z =   -33.800  mm,
	W =   -31.948 deg,	P =   -15.141 deg,	R =   -17.031 deg
   GP2:
	UF : 1, UT : 1,
	J1=    90.000 deg,	J2=   100.000 deg
};
P[449]{
   GP1:
	UF : 1, UT : 1,		CONFIG : 'N U T, 0, 0, 0',
	X =  2394.846  mm,	Y =   -83.445  mm,	Z =   -32.390  mm,
	W =   -31.930 deg,	P =   -15.141 deg,	R =   -17.037 deg
   GP2:
	UF : 1, UT : 1,
	J1=    90.000 deg,	J2=   100.000 deg
};
P[450]{
   GP1:
	UF : 1, UT : 1,		CONFIG : 'N U T, 0, 0, 0',
	X =  2420.835  mm,	Y =   -83.306  mm,	Z =   -29.423  mm,
	W =   -24.232 deg,	P =   -24.716 deg,	R =   -17.035 deg
   GP2:
	UF : 1, UT : 1,
	J1=    90.000 deg,	J2=   100.000 deg
};
P[451]{
   GP1:
	UF : 1, UT : 1,		CONFIG : 'N U T, 0, 0, 0',
	X =  2562.114  mm,	Y =  -708.403  mm,	Z =     7.893  mm,
	W =   -27.687 deg,	P =   -22.321 deg,	R =    54.103 deg
   GP2:
	UF : 1, UT : 1,
	J1=    80.000 deg,	J2=    90.000 deg
};
P[452]{
   GP1:
	UF : 1, UT : 1,		CONFIG : 'N U T, 0, 0, 0',
	X =  2517.838  mm,	Y =  -811.403  mm,	Z =     7.893  mm,
	W =   -27.687 deg,	P =   -22.321 deg,	R =    54.103 deg
   GP2:
	UF : 1, UT : 1,
	J1=    80.000 deg,	J2=    90.000 deg
};
P[453]{
   GP1:
	UF : 1, UT : 1,		CONFIG : 'N U T, 0, 0, -1',
	X =  2129.658  mm,	Y =   151.797  mm,	Z =   832.903  mm,
	W =     2.981 deg,	P =    35.499 deg,	R =   160.128 deg
   GP2:
	UF : 1, UT : 1,
	J1=    90.000 deg,	J2=    90.000 deg
};
P[454]{
   GP1:
	UF : 1, UT : 1,		CONFIG : 'N U T, 0, 0, -1',
	X =  2137.350  mm,	Y =   177.465  mm,	Z =   833.508  mm,
	W =     2.985 deg,	P =    35.513 deg,	R =   160.120 deg
   GP2:
	UF : 1, UT : 1,
	J1=    90.000 deg,	J2=    90.000 deg
};
P[455]{
   GP1:
	UF : 1, UT : 1,		CONFIG : 'N U T, 0, 0, 0',
	X =  2130.020  mm,	Y =   199.847  mm,	Z =   830.984  mm,
	W =     2.986 deg,	P =    35.518 deg,	R =  -100.169 deg
   GP2:
	UF : 1, UT : 1,
	J1=    90.000 deg,	J2=    90.000 deg
};
P[456]{
   GP1:
	UF : 1, UT : 1,		CONFIG : 'N U T, 0, 0, 0',
	X =  2102.832  mm,	Y =   191.069  mm,	Z =   829.130  mm,
	W =     2.988 deg,	P =    35.514 deg,	R =   -13.075 deg
   GP2:
	UF : 1, UT : 1,
	J1=    90.000 deg,	J2=    90.000 deg
};
P[457]{
   GP1:
	UF : 1, UT : 1,		CONFIG : 'N U T, 0, 0, 0',
	X =  2088.170  mm,	Y =   149.785  mm,	Z =   828.888  mm,
	W =     2.984 deg,	P =    35.513 deg,	R =   -13.072 deg
   GP2:
	UF : 1, UT : 1,
	J1=    90.000 deg,	J2=    90.000 deg
};
P[458]{
   GP1:
	UF : 1, UT : 1,		CONFIG : 'N U T, 0, 0, 0',
	X =  2102.574  mm,	Y =   126.514  mm,	Z =   830.669  mm,
	W =     2.985 deg,	P =    35.513 deg,	R =    80.476 deg
   GP2:
	UF : 1, UT : 1,
	J1=    90.000 deg,	J2=    90.000 deg
};
P[459]{
   GP1:
	UF : 1, UT : 1,		CONFIG : 'N U T, 0, 0, 0',
	X =  2551.662  mm,	Y =  -712.821  mm,	Z =   124.119  mm,
	W =   -35.203 deg,	P =   -31.584 deg,	R =    53.410 deg
   GP2:
	UF : 1, UT : 1,
	J1=    80.000 deg,	J2=    90.000 deg
};
P[460]{
   GP1:
	UF : 1, UT : 1,		CONFIG : 'N U T, 0, 0, 0',
	X =  1870.645  mm,	Y =  -712.821  mm,	Z =   348.203  mm,
	W =   -35.203 deg,	P =   -31.584 deg,	R =    53.410 deg
   GP2:
	UF : 1, UT : 1,
	J1=    80.000 deg,	J2=    90.000 deg
};
P[461]{
   GP1:
	UF : 1, UT : 1,		CONFIG : 'N U T, 0, 0, 0',
	X =   472.370  mm,	Y = -1534.903  mm,	Z =   492.380  mm,
	W =    50.539 deg,	P =     3.993 deg,	R =   -65.902 deg
   GP2:
	UF : 1, UT : 1,
	J1=    80.000 deg,	J2=    90.000 deg
};
P[462]{
   GP1:
	UF : 1, UT : 1,		CONFIG : 'N U T, 0, 0, 0',
	X =  2126.850  mm,	Y =   136.271  mm,	Z =   831.455  mm,
	W =     2.984 deg,	P =    35.513 deg,	R =   159.523 deg
   GP2:
	UF : 1, UT : 1,
	J1=    90.000 deg,	J2=    90.000 deg
};
P[463]{
   GP1:
	UF : 1, UT : 1,		CONFIG : 'N U T, 0, 0, 0',
	X =  2131.899  mm,	Y =   151.648  mm,	Z =   831.455  mm,
	W =     2.984 deg,	P =    35.513 deg,	R =   159.523 deg
   GP2:
	UF : 1, UT : 1,
	J1=    90.000 deg,	J2=    90.000 deg
};
P[464]{
   GP1:
	UF : 1, UT : 1,		CONFIG : 'N U T, 0, 0, 0',
	X =  2112.924  mm,	Y =   226.875  mm,	Z =   829.785  mm,
	W =    -2.360 deg,	P =    42.843 deg,	R =    86.536 deg
   GP2:
	UF : 1, UT : 1,
	J1=    90.000 deg,	J2=    90.000 deg
};
P[465]{
   GP1:
	UF : 1, UT : 1,		CONFIG : 'N U T, 0, 0, 0',
	X =  2202.613  mm,	Y =   227.153  mm,	Z =   829.824  mm,
	W =    -2.356 deg,	P =    42.846 deg,	R =    86.538 deg
   GP2:
	UF : 1, UT : 1,
	J1=    90.000 deg,	J2=    90.000 deg
};
P[466]{
   GP1:
	UF : 1, UT : 1,		CONFIG : 'N U T, 0, 0, 0',
	X =  2215.661  mm,	Y =   222.377  mm,	Z =   830.815  mm,
	W =    -2.493 deg,	P =    44.293 deg,	R =    56.655 deg
   GP2:
	UF : 1, UT : 1,
	J1=    90.000 deg,	J2=    90.000 deg
};
P[467]{
   GP1:
	UF : 1, UT : 1,		CONFIG : 'N U T, 0, 0, 0',
	X =  2222.874  mm,	Y =   213.385  mm,	Z =   828.313  mm,
	W =      .032 deg,	P =    44.143 deg,	R =    40.390 deg
   GP2:
	UF : 1, UT : 1,
	J1=    90.000 deg,	J2=    90.000 deg
};
P[468]{
   GP1:
	UF : 1, UT : 1,		CONFIG : 'N U T, 0, 0, 0',
	X =  2449.009  mm,	Y =   -44.468  mm,	Z =   827.867  mm,
	W =     -.128 deg,	P =    43.814 deg,	R =    45.335 deg
   GP2:
	UF : 1, UT : 1,
	J1=    90.000 deg,	J2=    90.000 deg
};
P[469]{
   GP1:
	UF : 1, UT : 1,		CONFIG : 'N U T, 0, 0, 0',
	X =  2612.111  mm,	Y = -1537.301  mm,	Z =  1175.202  mm,
	W =   -45.531 deg,	P =     6.252 deg,	R =    32.963 deg
   GP2:
	UF : 0, UT : 1,
	J1=   100.000 deg,	J2=   -90.000 deg
};
P[470]{
   GP1:
	UF : 1, UT : 1,		CONFIG : 'N U T, 0, 0, 0',
	X =  2071.007  mm,	Y = -1554.081  mm,	Z =  1677.384  mm,
	W =   -46.027 deg,	P =   -17.509 deg,	R =    23.991 deg
   GP2:
	UF : 1, UT : 1,
	J1=   100.000 deg,	J2=   -90.000 deg
};
P[471]{
   GP1:
	UF : 1, UT : 1,		CONFIG : 'N U T, 0, 0, 0',
	X =  1642.115  mm,	Y = -1225.593  mm,	Z =  1744.283  mm,
	W =   -30.785 deg,	P =   -19.925 deg,	R =    38.701 deg
   GP2:
	UF : 1, UT : 1,
	J1=   100.000 deg,	J2=   -90.000 deg
};
P[472]{
   GP1:
	UF : 1, UT : 1,		CONFIG : 'N U T, 0, 0, 0',
	X =  1044.179  mm,	Y =  -508.261  mm,	Z =   989.448  mm,
	W =    -7.948 deg,	P =   -16.175 deg,	R =    52.319 deg
   GP2:
	UF : 1, UT : 1,
	J1=   100.000 deg,	J2=   -90.000 deg
};
P[473]{
   GP1:
	UF : 1, UT : 1,		CONFIG : 'N U T, 0, 0, 0',
	X =  2659.725  mm,	Y =  1505.803  mm,	Z =  1079.609  mm,
	W =    15.908 deg,	P =   -31.536 deg,	R =   -26.500 deg
   GP2:
	UF : 0, UT : 1,
	J1=    95.000 deg,	J2=    90.000 deg
};
P[474]{
   GP1:
	UF : 1, UT : 1,		CONFIG : 'N U T, 0, 0, 0',
	X =  2454.781  mm,	Y =   -47.719  mm,	Z =   829.593  mm,
	W =      .165 deg,	P =    43.853 deg,	R =    54.355 deg
   GP2:
	UF : 1, UT : 1,
	J1=    90.000 deg,	J2=    90.000 deg
};
P[475]{
   GP1:
	UF : 1, UT : 1,		CONFIG : 'N U T, 0, 0, 0',
	X =  2459.541  mm,	Y =   -51.626  mm,	Z =   829.104  mm,
	W =    -1.320 deg,	P =    42.586 deg,	R =    55.587 deg
   GP2:
	UF : 1, UT : 1,
	J1=    90.000 deg,	J2=    90.000 deg
};
P[476]{
   GP1:
	UF : 1, UT : 1,		CONFIG : 'N U T, 0, 0, 0',
	X =  2655.978  mm,	Y =  -198.403  mm,	Z =   829.994  mm,
	W =   -30.974 deg,	P =    27.490 deg,	R =    12.667 deg
   GP2:
	UF : 1, UT : 1,
	J1=    90.000 deg,	J2=    90.000 deg
};
P[477]{
   GP1:
	UF : 1, UT : 1,		CONFIG : 'N U T, 0, 0, -1',
	X =  1225.021  mm,	Y = -1373.581  mm,	Z =   228.769  mm,
	W =   -54.518 deg,	P =     8.477 deg,	R =    24.180 deg
   GP2:
	UF : 1, UT : 1,
	J1=    90.000 deg,	J2=   -90.000 deg
};
P[478]{
   GP1:
	UF : 1, UT : 1,		CONFIG : 'N U T, 0, 0, -1',
	X =  2082.302  mm,	Y = -1064.969  mm,	Z =   253.594  mm,
	W =   -44.935 deg,	P =    -7.056 deg,	R =    83.172 deg
   GP2:
	UF : 1, UT : 1,
	J1=    90.000 deg,	J2=   -90.000 deg
};
P[479]{
   GP1:
	UF : 1, UT : 1,		CONFIG : 'N U T, 0, 0, -1',
	X =  2341.243  mm,	Y =  -989.972  mm,	Z =   103.893  mm,
	W =   -44.578 deg,	P =    -6.914 deg,	R =    83.049 deg
   GP2:
	UF : 1, UT : 1,
	J1=    90.000 deg,	J2=   -90.000 deg
};
P[480]{
   GP1:
	UF : 1, UT : 1,		CONFIG : 'N U T, 0, 0, -1',
	X =  2449.739  mm,	Y =  -869.683  mm,	Z =    46.520  mm,
	W =   -44.665 deg,	P =    -6.870 deg,	R =    84.747 deg
   GP2:
	UF : 1, UT : 1,
	J1=    90.000 deg,	J2=   -90.000 deg
};
P[481]{
   GP1:
	UF : 1, UT : 1,		CONFIG : 'N U T, 0, 0, 0',
	X =  2672.856  mm,	Y =  -207.422  mm,	Z =   831.831  mm,
	W =   -30.972 deg,	P =    27.486 deg,	R =    12.662 deg
   GP2:
	UF : 1, UT : 1,
	J1=    90.000 deg,	J2=    90.000 deg
};
P[482]{
   GP1:
	UF : 1, UT : 1,		CONFIG : 'N U T, 0, 0, 0',
	X =  2073.851  mm,	Y =    35.924  mm,	Z =    12.285  mm,
	W =   -30.951 deg,	P =    -2.135 deg,	R =   142.491 deg
   GP2:
	UF : 1, UT : 1,
	J1=    80.000 deg,	J2=    90.000 deg
};
P[483]{
   GP1:
	UF : 1, UT : 1,		CONFIG : 'N U T, 0, 0, 0',
	X =  2388.903  mm,	Y =  -813.009  mm,	Z =   289.336  mm,
	W =   -74.527 deg,	P =    19.606 deg,	R =   116.637 deg
   GP2:
	UF : 1, UT : 1,
	J1=    90.000 deg,	J2=   -90.000 deg
};
P[484]{
   GP1:
	UF : 1, UT : 1,		CONFIG : 'N U T, 0, 0, 0',
	X =  2319.444  mm,	Y =  -496.566  mm,	Z =   203.241  mm,
	W =    16.540 deg,	P =   -14.582 deg,	R =      .664 deg
   GP2:
	UF : 1, UT : 1,
	J1=    90.000 deg,	J2=   -90.000 deg
};
P[485]{
   GP1:
	UF : 1, UT : 1,		CONFIG : 'N U T, 0, 0, -1',
	X =  2429.174  mm,	Y =  -689.084  mm,	Z =   108.498  mm,
	W =   -41.825 deg,	P =    18.388 deg,	R =    51.054 deg
   GP2:
	UF : 1, UT : 1,
	J1=    90.000 deg,	J2=   -90.000 deg
};
P[486]{
   GP1:
	UF : 1, UT : 1,		CONFIG : 'N U T, 0, 0, 0',
	X =  2117.748  mm,	Y =    -4.566  mm,	Z =     3.630  mm,
	W =   -28.504 deg,	P =     6.349 deg,	R =   142.803 deg
   GP2:
	UF : 1, UT : 1,
	J1=    80.000 deg,	J2=    90.000 deg
};
P[487]{
   GP1:
	UF : 1, UT : 1,		CONFIG : 'N U T, 0, 0, 0',
	X =  2124.001  mm,	Y =   -12.191  mm,	Z =     2.432  mm,
	W =   -27.562 deg,	P =     5.114 deg,	R =   139.578 deg
   GP2:
	UF : 1, UT : 1,
	J1=    80.000 deg,	J2=    90.000 deg
};
P[488]{
   GP1:
	UF : 1, UT : 1,		CONFIG : 'N U T, 0, 0, 0',
	X =  2431.074  mm,	Y =  -699.084  mm,	Z =   106.298  mm,
	W =   -41.825 deg,	P =    18.388 deg,	R =    51.054 deg
   GP2:
	UF : 1, UT : 1,
	J1=    90.000 deg,	J2=   -90.000 deg
};
P[489]{
   GP1:
	UF : 1, UT : 1,		CONFIG : 'N U T, 0, 0, 0',
	X =  2429.174  mm,	Y =  -689.084  mm,	Z =   254.213  mm,
	W =   -57.120 deg,	P =     5.483 deg,	R =    47.853 deg
   GP2:
	UF : 1, UT : 1,
	J1=    90.000 deg,	J2=   -90.000 deg
};
P[490]{
   GP1:
	UF : 1, UT : 1,		CONFIG : 'N U T, 0, 0, 0',
	X =  1400.602  mm,	Y =  -689.084  mm,	Z =   254.213  mm,
	W =   -57.120 deg,	P =     5.483 deg,	R =    47.853 deg
   GP2:
	UF : 1, UT : 1,
	J1=    90.000 deg,	J2=   -90.000 deg
};
P[491]{
   GP1:
	UF : 1, UT : 1,		CONFIG : 'N U T, 0, 0, 0',
	X =  1400.602  mm,	Y =  -353.084  mm,	Z =   501.233  mm,
	W =    -2.074 deg,	P =   -10.233 deg,	R =    32.173 deg
   GP2:
	UF : 1, UT : 1,
	J1=    90.000 deg,	J2=  -135.000 deg
};
P[492]{
   GP1:
	UF : 1, UT : 1,		CONFIG : 'N U T, 0, 0, 0',
	X =  2655.602  mm,	Y =  -166.084  mm,	Z =   342.233  mm,
	W =     1.417 deg,	P =   -10.343 deg,	R =    12.808 deg
   GP2:
	UF : 1, UT : 1,
	J1=    90.000 deg,	J2=  -135.000 deg
};
P[493]{
   GP1:
	UF : 1, UT : 1,		CONFIG : 'N U T, 0, 0, 0',
	X =  2130.131  mm,	Y =   -20.247  mm,	Z =     1.791  mm,
	W =   -27.580 deg,	P =     5.122 deg,	R =   136.990 deg
   GP2:
	UF : 1, UT : 1,
	J1=    80.000 deg,	J2=    90.000 deg
};
P[494]{
   GP1:
	UF : 1, UT : 1,		CONFIG : 'N U T, 0, 0, 0',
	X =  2586.641  mm,	Y =  1526.023  mm,	Z =  1082.786  mm,
	W =    42.689 deg,	P =    16.599 deg,	R =   -42.374 deg
   GP2:
	UF : 0, UT : 1,
	J1=    95.000 deg,	J2=    90.000 deg
};
P[495]{
   GP1:
	UF : 1, UT : 1,		CONFIG : 'N U T, 0, 0, 0',
	X =  2823.448  mm,	Y =  -159.890  mm,	Z =   258.839  mm,
	W =    -7.346 deg,	P =   -29.104 deg,	R =    14.845 deg
   GP2:
	UF : 1, UT : 1,
	J1=    90.000 deg,	J2=  -135.000 deg
};
P[496]{
   GP1:
	UF : 1, UT : 1,		CONFIG : 'N U T, 0, 0, 0',
	X =  2357.965  mm,	Y =  -270.302  mm,	Z =   258.839  mm,
	W =    -1.017 deg,	P =    -4.421 deg,	R =    12.975 deg
   GP2:
	UF : 1, UT : 1,
	J1=    90.000 deg,	J2=  -135.000 deg
};
P[497]{
   GP1:
	UF : 1, UT : 1,		CONFIG : 'N U T, 0, 0, 0',
	X =  1536.098  mm,	Y =  1365.318  mm,	Z =  1433.705  mm,
	W =    42.689 deg,	P =    16.599 deg,	R =   -30.305 deg
   GP2:
	UF : 1, UT : 1,
	J1=    95.000 deg,	J2=    90.000 deg
};
P[498]{
   GP1:
	UF : 1, UT : 1,		CONFIG : 'N U T, 0, 0, 0',
	X =   498.430  mm,	Y =  -249.509  mm,	Z =  2387.961  mm,
	W =     2.736 deg,	P =   -33.821 deg,	R =   -22.668 deg
   GP2:
	UF : 1, UT : 1,
	J1=    80.000 deg,	J2=    90.000 deg
};
P[499]{
   GP1:
	UF : 1, UT : 1,		CONFIG : 'N U T, 0, 0, 0',
	X =  2641.832  mm,	Y =  -264.435  mm,	Z =   263.645  mm,
	W =     0.000 deg,	P =    -6.880 deg,	R =    -2.940 deg
   GP2:
	UF : 1, UT : 1,
	J1=    90.000 deg,	J2=  -135.000 deg
};
P[500]{
   GP1:
	UF : 1, UT : 1,		CONFIG : 'N U T, 0, 0, 0',
	X =  2474.831  mm,	Y =   -41.435  mm,	Z =    90.241  mm,
	W =    43.945 deg,	P =   -11.174 deg,	R =     1.639 deg
   GP2:
	UF : 1, UT : 1,
	J1=    90.000 deg,	J2=   -90.000 deg
};
P[501]{
   GP1:
	UF : 1, UT : 1,		CONFIG : 'N U T, 0, 0, 0',
	X =  2474.831  mm,	Y =    90.943  mm,	Z =    79.910  mm,
	W =    39.708 deg,	P =   -23.339 deg,	R =    15.773 deg
   GP2:
	UF : 1, UT : 1,
	J1=    90.000 deg,	J2=   -90.000 deg
};
P[502]{
   GP1:
	UF : 1, UT : 1,		CONFIG : 'N U T, 0, 0, 0',
	X =  1773.758  mm,	Y =  1132.590  mm,	Z =   293.935  mm,
	W =   -17.776 deg,	P =    15.458 deg,	R =    47.254 deg
   GP2:
	UF : 1, UT : 1,
	J1=    90.000 deg,	J2=    90.000 deg
};
P[503]{
   GP1:
	UF : 1, UT : 1,		CONFIG : 'N U T, 0, 0, -1',
	X =  1391.376  mm,	Y = -1411.270  mm,	Z =  1335.234  mm,
	W =   -82.179 deg,	P =     1.788 deg,	R =    24.906 deg
   GP2:
	UF : 1, UT : 1,
	J1=    90.000 deg,	J2=   -90.000 deg
};
P[504]{
   GP1:
	UF : 1, UT : 1,		CONFIG : 'N U B, 0, 0, 0',
	X =   357.030  mm,	Y =     -.134  mm,	Z =  2422.493  mm,
	W =     -.020 deg,	P =   -39.773 deg,	R =      .020 deg
   GP2:
	UF : 1, UT : 1,
	J1=    90.000 deg,	J2=    90.000 deg
};
P[505]{
   GP1:
	UF : 1, UT : 1,		CONFIG : 'N U T, 0, 0, 0',
	X =  2478.831  mm,	Y =    82.943  mm,	Z =    74.910  mm,
	W =    39.708 deg,	P =   -23.339 deg,	R =    15.773 deg
   GP2:
	UF : 1, UT : 1,
	J1=    90.000 deg,	J2=   -90.000 deg
};
P[506]{
   GP1:
	UF : 1, UT : 1,		CONFIG : 'N U T, 0, 0, 0',
	X =  2474.831  mm,	Y =  -180.721  mm,	Z =    90.242  mm,
	W =    43.034 deg,	P =    14.904 deg,	R =   -25.132 deg
   GP2:
	UF : 1, UT : 1,
	J1=    90.000 deg,	J2=   -90.000 deg
};
P[507]{
   GP1:
	UF : 1, UT : 1,		CONFIG : 'N U T, 0, 0, 0',
	X =  1656.260  mm,	Y =  -180.721  mm,	Z =    90.242  mm,
	W =    43.034 deg,	P =    14.904 deg,	R =   -25.132 deg
   GP2:
	UF : 1, UT : 1,
	J1=    90.000 deg,	J2=   -90.000 deg
};
P[508]{
   GP1:
	UF : 1, UT : 1,		CONFIG : 'N U B, 0, 0, 0',
	X =   357.030  mm,	Y =     -.134  mm,	Z =  2422.493  mm,
	W =     -.020 deg,	P =   -39.773 deg,	R =      .020 deg
   GP2:
	UF : 1, UT : 1,
	J1=    90.000 deg,	J2=   -90.000 deg
};
P[509]{
   GP1:
	UF : 1, UT : 1,		CONFIG : 'N U T, 0, 0, 0',
	X =  2251.754  mm,	Y =  -187.747  mm,	Z =   -18.626  mm,
	W =   -36.464 deg,	P =    -8.806 deg,	R =   122.583 deg
   GP2:
	UF : 1, UT : 1,
	J1=    80.000 deg,	J2=    90.000 deg
};
P[510]{
   GP1:
	UF : 1, UT : 1,		CONFIG : 'N U T, 0, 0, 0',
	X =  2260.659  mm,	Y =  -197.463  mm,	Z =   -20.538  mm,
	W =   -36.554 deg,	P =   -11.684 deg,	R =   125.973 deg
   GP2:
	UF : 1, UT : 1,
	J1=    80.000 deg,	J2=    90.000 deg
};
P[511]{
   GP1:
	UF : 1, UT : 1,		CONFIG : 'N U T, 0, 0, 0',
	X =  2269.185  mm,	Y =  -206.886  mm,	Z =   -21.960  mm,
	W =   -36.304 deg,	P =   -14.510 deg,	R =   128.303 deg
   GP2:
	UF : 1, UT : 1,
	J1=    80.000 deg,	J2=    90.000 deg
};
P[512]{
   GP1:
	UF : 1, UT : 1,		CONFIG : 'N U T, 0, 0, 0',
	X =  2511.863  mm,	Y =  -435.567  mm,	Z =   -65.547  mm,
	W =   -23.381 deg,	P =   -31.779 deg,	R =    95.136 deg
   GP2:
	UF : 1, UT : 1,
	J1=    80.000 deg,	J2=    90.000 deg
};
P[513]{
   GP1:
	UF : 1, UT : 1,		CONFIG : 'N U T, 0, 0, 0',
	X =  2535.927  mm,	Y =  -449.078  mm,	Z =   -69.737  mm,
	W =   -18.431 deg,	P =   -37.735 deg,	R =   100.755 deg
   GP2:
	UF : 1, UT : 1,
	J1=    80.000 deg,	J2=    90.000 deg
};
P[514]{
   GP1:
	UF : 1, UT : 1,		CONFIG : 'N U T, 0, 0, 0',
	X =  2558.091  mm,	Y =  -453.543  mm,	Z =   -73.418  mm,
	W =   -18.771 deg,	P =   -39.987 deg,	R =   104.546 deg
   GP2:
	UF : 1, UT : 1,
	J1=    80.000 deg,	J2=    90.000 deg
};
P[515]{
   GP1:
	UF : 1, UT : 1,		CONFIG : 'N U T, 0, 0, 0',
	X =  2574.982  mm,	Y =  -457.797  mm,	Z =   -77.599  mm,
	W =   -22.267 deg,	P =   -37.927 deg,	R =   106.779 deg
   GP2:
	UF : 1, UT : 1,
	J1=    80.000 deg,	J2=    90.000 deg
};
P[516]{
   GP1:
	UF : 1, UT : 1,		CONFIG : 'N U T, 0, 0, 0',
	X =  2621.992  mm,	Y =  -529.847  mm,	Z =   -85.920  mm,
	W =   -33.012 deg,	P =   -16.164 deg,	R =    66.999 deg
   GP2:
	UF : 1, UT : 1,
	J1=    80.000 deg,	J2=    90.000 deg
};
P[517]{
   GP1:
	UF : 1, UT : 1,		CONFIG : 'N U T, 0, 0, 0',
	X =  2621.958  mm,	Y =  -548.775  mm,	Z =   -86.023  mm,
	W =   -33.009 deg,	P =   -16.162 deg,	R =    66.994 deg
   GP2:
	UF : 1, UT : 1,
	J1=    80.000 deg,	J2=    90.000 deg
};
P[518]{
   GP1:
	UF : 1, UT : 1,		CONFIG : 'N U T, 0, 0, 0',
	X =  2620.833  mm,	Y =  -724.953  mm,	Z =   -86.008  mm,
	W =   -27.674 deg,	P =   -22.322 deg,	R =    54.091 deg
   GP2:
	UF : 1, UT : 1,
	J1=    80.000 deg,	J2=    90.000 deg
};
P[519]{
   GP1:
	UF : 1, UT : 1,		CONFIG : 'N U T, 0, 0, 0',
	X =  1477.103  mm,	Y =  -165.683  mm,	Z =   137.951  mm,
	W =    38.761 deg,	P =    24.667 deg,	R =   -44.781 deg
   GP2:
	UF : 1, UT : 1,
	J1=    90.000 deg,	J2=   -90.000 deg
};
P[520]{
   GP1:
	UF : 1, UT : 1,		CONFIG : 'N U T, 0, 0, 0',
	X =  2334.769  mm,	Y =  -176.256  mm,	Z =   129.823  mm,
	W =    49.996 deg,	P =    12.253 deg,	R =   -42.841 deg
   GP2:
	UF : 1, UT : 1,
	J1=    90.000 deg,	J2=   -90.000 deg
};
P[521]{
   GP1:
	UF : 1, UT : 1,		CONFIG : 'N U T, 0, 0, 0',
	X =  2334.769  mm,	Y =    95.744  mm,	Z =   109.147  mm,
	W =    41.080 deg,	P =   -17.089 deg,	R =    29.592 deg
   GP2:
	UF : 1, UT : 1,
	J1=    90.000 deg,	J2=   -90.000 deg
};
P[522]{
   GP1:
	UF : 1, UT : 1,		CONFIG : 'N U T, 0, 0, 0',
	X =  2550.739  mm,	Y =  -832.902  mm,	Z =   -76.728  mm,
	W =   -27.690 deg,	P =   -22.316 deg,	R =    54.107 deg
   GP2:
	UF : 1, UT : 1,
	J1=    80.000 deg,	J2=    90.000 deg
};
P[523]{
   GP1:
	UF : 1, UT : 1,		CONFIG : 'N U T, 0, 0, 0',
	X =  2551.660  mm,	Y =  -813.166  mm,	Z =   -76.438  mm,
	W =   -27.682 deg,	P =   -22.308 deg,	R =    54.092 deg
   GP2:
	UF : 1, UT : 1,
	J1=    80.000 deg,	J2=    90.000 deg
};
P[524]{
   GP1:
	UF : 1, UT : 1,		CONFIG : 'N U T, 0, 0, 0',
	X =  2565.317  mm,	Y =  -801.232  mm,	Z =   -77.060  mm,
	W =   -27.686 deg,	P =   -22.321 deg,	R =    23.348 deg
   GP2:
	UF : 1, UT : 1,
	J1=    80.000 deg,	J2=    90.000 deg
};
P[525]{
   GP1:
	UF : 1, UT : 1,		CONFIG : 'N U T, 0, 0, 0',
	X =  2340.804  mm,	Y =    96.102  mm,	Z =    56.984  mm,
	W =    34.887 deg,	P =   -26.988 deg,	R =    21.909 deg
   GP2:
	UF : 1, UT : 1,
	J1=    90.000 deg,	J2=   -90.000 deg
};
P[526]{
   GP1:
	UF : 1, UT : 1,		CONFIG : 'N U T, 0, 0, 0',
	X =  2334.769  mm,	Y =  -176.256  mm,	Z =   129.823  mm,
	W =    49.996 deg,	P =    12.253 deg,	R =   -42.841 deg
   GP2:
	UF : 1, UT : 1,
	J1=    90.000 deg,	J2=   -90.000 deg
};
P[527]{
   GP1:
	UF : 1, UT : 1,		CONFIG : 'N U T, 0, 0, 0',
	X =  1274.769  mm,	Y =  -176.256  mm,	Z =   129.823  mm,
	W =    14.633 deg,	P =    39.206 deg,	R =   -59.040 deg
   GP2:
	UF : 1, UT : 1,
	J1=    90.000 deg,	J2=   -90.000 deg
};
P[528]{
   GP1:
	UF : 1, UT : 1,		CONFIG : 'N U T, 0, 0, 0',
	X =  1137.626  mm,	Y =   231.744  mm,	Z =   129.823  mm,
	W =     5.452 deg,	P =    45.384 deg,	R =    96.559 deg
   GP2:
	UF : 1, UT : 1,
	J1=    90.000 deg,	J2=   -90.000 deg
};
P[529]{
   GP1:
	UF : 1, UT : 1,		CONFIG : 'N U T, 0, 0, 0',
	X =  1702.626  mm,	Y =   216.744  mm,	Z =    45.395  mm,
	W =   -35.057 deg,	P =    31.336 deg,	R =    18.229 deg
   GP2:
	UF : 1, UT : 1,
	J1=    90.000 deg,	J2=   -90.000 deg
};
P[530]{
   GP1:
	UF : 1, UT : 1,		CONFIG : 'N U T, 0, 0, 0',
	X =  2576.762  mm,	Y =  -796.353  mm,	Z =   -82.224  mm,
	W =   -33.350 deg,	P =   -11.305 deg,	R =    17.629 deg
   GP2:
	UF : 1, UT : 1,
	J1=    80.000 deg,	J2=    90.000 deg
};
P[531]{
   GP1:
	UF : 1, UT : 1,		CONFIG : 'N U T, 0, 0, 0',
	X =  2611.385  mm,	Y =  -766.607  mm,	Z =   -84.979  mm,
	W =   -30.071 deg,	P =    -4.704 deg,	R =    42.986 deg
   GP2:
	UF : 1, UT : 1,
	J1=    80.000 deg,	J2=    90.000 deg
};
P[532]{
   GP1:
	UF : 1, UT : 1,		CONFIG : 'N U T, 0, 0, 0',
	X =  2624.754  mm,	Y =  -718.507  mm,	Z =   -86.108  mm,
	W =   -25.591 deg,	P =   -24.735 deg,	R =    48.858 deg
   GP2:
	UF : 1, UT : 1,
	J1=    80.000 deg,	J2=    90.000 deg
};
P[533]{
   GP1:
	UF : 1, UT : 1,		CONFIG : 'N U T, 0, 0, -1',
	X =  2494.854  mm,	Y =  -857.680  mm,	Z =    -8.806  mm,
	W =   -44.580 deg,	P =    -6.907 deg,	R =    84.735 deg
   GP2:
	UF : 1, UT : 1,
	J1=    90.000 deg,	J2=   -90.000 deg
};
P[534]{
   GP1:
	UF : 1, UT : 1,		CONFIG : 'N U T, 0, 0, 0',
	X =  1968.756  mm,	Y =   235.799  mm,	Z =    41.294  mm,
	W =   -37.049 deg,	P =    22.562 deg,	R =    41.911 deg
   GP2:
	UF : 1, UT : 1,
	J1=    90.000 deg,	J2=   -90.000 deg
};
P[535]{
   GP1:
	UF : 1, UT : 1,		CONFIG : 'N U T, 0, 0, 0',
	X =  2281.156  mm,	Y =   263.463  mm,	Z =    29.688  mm,
	W =   -37.041 deg,	P =    22.569 deg,	R =    41.916 deg
   GP2:
	UF : 1, UT : 1,
	J1=    83.000 deg,	J2=   -90.000 deg
};
P[536]{
   GP1:
	UF : 1, UT : 1,		CONFIG : 'N U T, 0, 0, 0',
	X =  2487.498  mm,	Y =   206.111  mm,	Z =    13.958  mm,
	W =   -43.230 deg,	P =      .800 deg,	R =   -58.961 deg
   GP2:
	UF : 1, UT : 1,
	J1=    83.000 deg,	J2=   -90.000 deg
};
P[537]{
   GP1:
	UF : 1, UT : 1,		CONFIG : 'N U T, 0, 0, 0',
	X =  2487.758  mm,	Y =   132.800  mm,	Z =    41.293  mm,
	W =   -42.488 deg,	P =     1.841 deg,	R =   -72.344 deg
   GP2:
	UF : 1, UT : 1,
	J1=    83.000 deg,	J2=   -90.000 deg
};
P[538]{
   GP1:
	UF : 1, UT : 1,		CONFIG : 'N U T, 0, 0, -1',
	X =  2494.926  mm,	Y =  -777.781  mm,	Z =    -9.320  mm,
	W =   -44.580 deg,	P =    -6.907 deg,	R =    84.735 deg
   GP2:
	UF : 1, UT : 1,
	J1=    90.000 deg,	J2=   -90.000 deg
};
P[539]{
   GP1:
	UF : 1, UT : 1,		CONFIG : 'N U T, 0, 0, 0',
	X =  2518.619  mm,	Y =  -755.627  mm,	Z =    -6.486  mm,
	W =   -39.981 deg,	P =    14.824 deg,	R =    17.712 deg
   GP2:
	UF : 1, UT : 1,
	J1=    90.000 deg,	J2=   -90.000 deg
};
P[540]{
   GP1:
	UF : 1, UT : 1,		CONFIG : 'N U T, 0, 0, 0',
	X =  2567.877  mm,	Y =  -756.992  mm,	Z =    -7.047  mm,
	W =   -39.981 deg,	P =    14.824 deg,	R =    17.712 deg
   GP2:
	UF : 1, UT : 1,
	J1=    90.000 deg,	J2=   -90.000 deg
};
P[541]{
   GP1:
	UF : 1, UT : 1,		CONFIG : 'N U T, 0, 0, 0',
	X =  2752.964  mm,	Y =  -168.876  mm,	Z =   176.244  mm,
	W =    -1.647 deg,	P =    -7.143 deg,	R =    13.032 deg
   GP2:
	UF : 1, UT : 1,
	J1=    90.000 deg,	J2=  -135.000 deg
};
P[542]{
   GP1:
	UF : 1, UT : 1,		CONFIG : 'N U T, 0, 0, 0',
	X =  2487.758  mm,	Y =   132.800  mm,	Z =    41.293  mm,
	W =   -42.488 deg,	P =     1.841 deg,	R =   -72.344 deg
   GP2:
	UF : 1, UT : 1,
	J1=    83.000 deg,	J2=   -90.000 deg
};
P[543]{
   GP1:
	UF : 1, UT : 1,		CONFIG : 'N U T, 0, 0, 0',
	X =  2487.757  mm,	Y =   235.800  mm,	Z =    41.293  mm,
	W =   -46.494 deg,	P =   -14.946 deg,	R =     1.465 deg
   GP2:
	UF : 1, UT : 1,
	J1=    83.000 deg,	J2=   -90.000 deg
};
P[544]{
   GP1:
	UF : 1, UT : 1,		CONFIG : 'N U T, 0, 0, 0',
	X =  2363.757  mm,	Y =   235.799  mm,	Z =    47.485  mm,
	W =   -46.494 deg,	P =   -14.946 deg,	R =     1.465 deg
   GP2:
	UF : 1, UT : 1,
	J1=    90.000 deg,	J2=   -90.000 deg
};
P[545]{
   GP1:
	UF : 1, UT : 1,		CONFIG : 'N U T, 0, 0, 0',
	X =  2865.942  mm,	Y =  -168.094  mm,	Z =   177.218  mm,
	W =    -5.450 deg,	P =   -22.504 deg,	R =    14.017 deg
   GP2:
	UF : 1, UT : 1,
	J1=    90.000 deg,	J2=  -135.000 deg
};
P[546]{
   GP1:
	UF : 1, UT : 1,		CONFIG : 'N U T, 0, 0, 0',
	X =  2379.984  mm,	Y =  -271.988  mm,	Z =    87.998  mm,
	W =      .003 deg,	P =      .001 deg,	R =    -2.945 deg
   GP2:
	UF : 1, UT : 1,
	J1=    90.000 deg,	J2=  -135.000 deg
};
P[547]{
   GP1:
	UF : 1, UT : 1,		CONFIG : 'N U T, 0, 0, 0',
	X =  2483.422  mm,	Y =   242.950  mm,	Z =    62.981  mm,
	W =   -44.990 deg,	P =    -1.038 deg,	R =    17.559 deg
   GP2:
	UF : 1, UT : 1,
	J1=    90.000 deg,	J2=   -90.000 deg
};
P[548]{
   GP1:
	UF : 1, UT : 1,		CONFIG : 'N U T, 0, 0, 0',
	X =  2280.422  mm,	Y =   242.950  mm,	Z =    62.981  mm,
	W =   -44.990 deg,	P =    -1.038 deg,	R =    17.559 deg
   GP2:
	UF : 1, UT : 1,
	J1=    90.000 deg,	J2=   -90.000 deg
};
P[549]{
   GP1:
	UF : 1, UT : 1,		CONFIG : 'N U T, 0, 0, 0',
	X =  2280.422  mm,	Y =   142.950  mm,	Z =    62.981  mm,
	W =   -44.990 deg,	P =    -1.038 deg,	R =    17.559 deg
   GP2:
	UF : 1, UT : 1,
	J1=    90.000 deg,	J2=   -90.000 deg
};
P[550]{
   GP1:
	UF : 1, UT : 1,		CONFIG : 'N U T, 0, 0, 0',
	X =  2755.499  mm,	Y =  -271.313  mm,	Z =    89.477  mm,
	W =      .076 deg,	P =    -1.495 deg,	R =    -2.941 deg
   GP2:
	UF : 1, UT : 1,
	J1=    90.000 deg,	J2=  -135.000 deg
};
P[551]{
   GP1:
	UF : 1, UT : 1,		CONFIG : 'N U T, 0, 0, 0',
	X =  2504.732  mm,	Y =   163.801  mm,	Z =    -7.840  mm,
	W =    37.870 deg,	P =   -26.386 deg,	R =    31.563 deg
   GP2:
	UF : 1, UT : 1,
	J1=    90.000 deg,	J2=   -90.000 deg
};
P[552]{
   GP1:
	UF : 1, UT : 1,		CONFIG : 'N U T, 0, 0, 0',
	X =  2464.249  mm,	Y =   164.384  mm,	Z =    -7.847  mm,
	W =    37.874 deg,	P =   -26.389 deg,	R =    31.563 deg
   GP2:
	UF : 1, UT : 1,
	J1=    90.000 deg,	J2=   -90.000 deg
};
P[553]{
   GP1:
	UF : 1, UT : 1,		CONFIG : 'N U T, 0, 0, 0',
	X =  2280.422  mm,	Y =   218.557  mm,	Z =   105.269  mm,
	W =   -44.990 deg,	P =    -1.038 deg,	R =    25.270 deg
   GP2:
	UF : 1, UT : 1,
	J1=    90.000 deg,	J2=   -90.000 deg
};
P[554]{
   GP1:
	UF : 1, UT : 1,		CONFIG : 'N U T, 0, 0, 0',
	X =  1204.422  mm,	Y =   218.557  mm,	Z =   105.269  mm,
	W =   -29.046 deg,	P =    29.449 deg,	R =    29.350 deg
   GP2:
	UF : 1, UT : 1,
	J1=    90.000 deg,	J2=   -90.000 deg
};
P[555]{
   GP1:
	UF : 1, UT : 1,		CONFIG : 'N U T, 0, 0, 0',
	X =  1204.422  mm,	Y =  -167.443  mm,	Z =  1122.269  mm,
	W =   -44.990 deg,	P =    -1.038 deg,	R =    25.270 deg
   GP2:
	UF : 1, UT : 1,
	J1=    90.000 deg,	J2=   -90.000 deg
};
P[556]{
   GP1:
	UF : 1, UT : 1,		CONFIG : 'N U T, 0, 0, 0',
	X =  2328.690  mm,	Y =   -25.109  mm,	Z =   925.961  mm,
	W =    38.029 deg,	P =    27.224 deg,	R =   -32.413 deg
   GP2:
	UF : 1, UT : 1,
	J1=    90.000 deg,	J2=   -90.000 deg
};
P[557]{
   GP1:
	UF : 1, UT : 1,		CONFIG : 'N U T, 0, 0, 0',
	X =  2444.114  mm,	Y =   163.873  mm,	Z =    -8.034  mm,
	W =    40.554 deg,	P =   -21.460 deg,	R =    53.231 deg
   GP2:
	UF : 1, UT : 1,
	J1=    90.000 deg,	J2=   -90.000 deg
};
P[558]{
   GP1:
	UF : 1, UT : 1,		CONFIG : 'N U T, 0, 0, 0',
	X =  1685.665  mm,	Y =   -64.872  mm,	Z =   -18.365  mm,
	W =    41.394 deg,	P =    19.519 deg,	R =   -17.046 deg
   GP2:
	UF : 1, UT : 1,
	J1=    90.000 deg,	J2=   -90.000 deg
};
P[559]{
   GP1:
	UF : 1, UT : 1,		CONFIG : 'N U T, 0, 0, 0',
	X =  2407.814  mm,	Y =    -3.230  mm,	Z =   914.873  mm,
	W =    36.706 deg,	P =    26.470 deg,	R =   -16.230 deg
   GP2:
	UF : 1, UT : 1,
	J1=    90.000 deg,	J2=   -90.000 deg
};
P[560]{
   GP1:
	UF : 1, UT : 1,		CONFIG : 'N U T, 0, 0, 0',
	X =  2432.823  mm,	Y =   104.215  mm,	Z =   863.805  mm,
	W =     4.851 deg,	P =    34.958 deg,	R =    24.131 deg
   GP2:
	UF : 1, UT : 1,
	J1=    89.999 deg,	J2=   -90.000 deg
};
P[561]{
   GP1:
	UF : 1, UT : 1,		CONFIG : 'N U T, 0, 0, 0',
	X =  1655.518  mm,	Y =   -66.180  mm,	Z =   -18.364  mm,
	W =    41.393 deg,	P =    19.514 deg,	R =   -16.107 deg
   GP2:
	UF : 1, UT : 1,
	J1=    90.000 deg,	J2=   -90.000 deg
};
P[562]{
   GP1:
	UF : 1, UT : 1,		CONFIG : 'N U T, 0, 0, 0',
	X =  1644.071  mm,	Y =   -64.443  mm,	Z =   -18.488  mm,
	W =    41.392 deg,	P =    19.514 deg,	R =     3.473 deg
   GP2:
	UF : 1, UT : 1,
	J1=    90.000 deg,	J2=   -90.000 deg
};
P[563]{
   GP1:
	UF : 1, UT : 1,		CONFIG : 'N U T, 0, 0, 0',
	X =  2459.632  mm,	Y =   122.370  mm,	Z =   906.747  mm,
	W =    -6.207 deg,	P =    17.663 deg,	R =    19.082 deg
   GP2:
	UF : 1, UT : 1,
	J1=    89.999 deg,	J2=   -90.000 deg
};
P[564]{
   GP1:
	UF : 1, UT : 1,		CONFIG : 'N U T, 0, 0, 0',
	X =  1677.456  mm,	Y = -1378.259  mm,	Z =  1040.445  mm,
	W =   -45.493 deg,	P =   -19.537 deg,	R =    48.719 deg
   GP2:
	UF : 1, UT : 1,
	J1=   180.000 deg,	J2=  -125.000 deg
};
P[565]{
   GP1:
	UF : 1, UT : 1,		CONFIG : 'N U T, 0, 0, 0',
	X =  2301.523  mm,	Y =   100.306  mm,	Z =   896.809  mm,
	W =   -38.032 deg,	P =    -5.730 deg,	R =    38.955 deg
   GP2:
	UF : 1, UT : 1,
	J1=    89.999 deg,	J2=   -90.000 deg
};
P[566]{
   GP1:
	UF : 1, UT : 1,		CONFIG : 'N U T, 0, 0, 0',
	X =  1635.702  mm,	Y =   -66.864  mm,	Z =   -17.244  mm,
	W =    41.392 deg,	P =    19.514 deg,	R =    24.112 deg
   GP2:
	UF : 1, UT : 1,
	J1=    90.000 deg,	J2=   -90.000 deg
};
P[567]{
   GP1:
	UF : 1, UT : 1,		CONFIG : 'N U T, 0, 0, 0',
	X =  1608.120  mm,	Y =   -97.236  mm,	Z =   -17.308  mm,
	W =    37.029 deg,	P =    27.659 deg,	R =    15.298 deg
   GP2:
	UF : 1, UT : 1,
	J1=    90.000 deg,	J2=   -90.000 deg
};
P[568]{
   GP1:
	UF : 1, UT : 1,		CONFIG : 'N U T, 0, 0, 0',
	X =  2343.829  mm,	Y =   125.019  mm,	Z =   873.736  mm,
	W =   -38.032 deg,	P =    -5.730 deg,	R =    38.955 deg
   GP2:
	UF : 1, UT : 1,
	J1=    89.999 deg,	J2=   -90.000 deg
};
P[569]{
   GP1:
	UF : 1, UT : 1,		CONFIG : 'N U T, 0, 0, 0',
	X =  1695.422  mm,	Y =   -78.871  mm,	Z =  1381.555  mm,
	W =    -4.515 deg,	P =      .965 deg,	R =    -2.729 deg
   GP2:
	UF : 1, UT : 1,
	J1=    90.000 deg,	J2=   -90.000 deg
};
P[570]{
   GP1:
	UF : 1, UT : 1,		CONFIG : 'N U T, 0, 0, 0',
	X =  1588.118  mm,	Y =  -108.567  mm,	Z =   -16.888  mm,
	W =    38.940 deg,	P =    23.604 deg,	R =   -29.723 deg
   GP2:
	UF : 1, UT : 1,
	J1=    90.000 deg,	J2=   -90.000 deg
};
P[571]{
   GP1:
	UF : 1, UT : 1,		CONFIG : 'N U T, 0, 0, 0',
	X =  1618.043  mm,	Y = -1395.782  mm,	Z =  1053.900  mm,
	W =   -44.560 deg,	P =   -18.266 deg,	R =    45.822 deg
   GP2:
	UF : 1, UT : 1,
	J1=   180.000 deg,	J2=  -125.000 deg
};
P[572]{
   GP1:
	UF : 1, UT : 1,		CONFIG : 'N U T, 0, 0, 0',
	X =  2106.244  mm,	Y =  -177.973  mm,	Z =   164.824  mm,
	W =    -4.184 deg,	P =     7.592 deg,	R =    43.674 deg
   GP2:
	UF : 1, UT : 1,
	J1=    90.000 deg,	J2=  -100.000 deg
};
P[573]{
   GP1:
	UF : 1, UT : 1,		CONFIG : 'N U T, 0, 0, 0',
	X =  2106.243  mm,	Y =   -20.258  mm,	Z =   164.824  mm,
	W =     2.218 deg,	P =    14.051 deg,	R =    70.281 deg
   GP2:
	UF : 1, UT : 1,
	J1=    90.000 deg,	J2=  -100.000 deg
};
P[574]{
   GP1:
	UF : 1, UT : 1,		CONFIG : 'N U T, 0, 0, 0',
	X =  1562.037  mm,	Y =   -85.294  mm,	Z =   -16.902  mm,
	W =    36.730 deg,	P =    28.082 deg,	R =  -109.081 deg
   GP2:
	UF : 1, UT : 1,
	J1=    90.000 deg,	J2=   -90.000 deg
};
P[575]{
   GP1:
	UF : 1, UT : 1,		CONFIG : 'N U T, 0, 0, 0',
	X =  1556.914  mm,	Y =   -40.647  mm,	Z =   -16.118  mm,
	W =    36.727 deg,	P =    28.082 deg,	R =  -114.509 deg
   GP2:
	UF : 1, UT : 1,
	J1=    90.000 deg,	J2=   -90.000 deg
};
P[576]{
   GP1:
	UF : 1, UT : 1,		CONFIG : 'N U T, 0, 0, 0',
	X =  2113.743  mm,	Y =   -23.258  mm,	Z =   164.824  mm,
	W =     2.218 deg,	P =    14.051 deg,	R =    70.281 deg
   GP2:
	UF : 1, UT : 1,
	J1=    90.000 deg,	J2=  -100.000 deg
};
P[577]{
   GP1:
	UF : 1, UT : 1,		CONFIG : 'N U T, 0, 0, 0',
	X =  2106.244  mm,	Y =  -177.973  mm,	Z =   164.824  mm,
	W =    -4.184 deg,	P =     7.592 deg,	R =    43.674 deg
   GP2:
	UF : 1, UT : 1,
	J1=    90.000 deg,	J2=  -100.000 deg
};
P[578]{
   GP1:
	UF : 1, UT : 1,		CONFIG : 'N U T, 0, 0, 0',
	X =  2154.661  mm,	Y =  -177.973  mm,	Z =   164.824  mm,
	W =    28.994 deg,	P =   -15.433 deg,	R =    30.441 deg
   GP2:
	UF : 1, UT : 1,
	J1=    90.000 deg,	J2=   -90.000 deg
};
P[579]{
   GP1:
	UF : 1, UT : 1,		CONFIG : 'N U T, 0, 0, 0',
	X =  1556.835  mm,	Y =   -36.070  mm,	Z =   -15.557  mm,
	W =    39.289 deg,	P =    28.081 deg,	R =   -80.638 deg
   GP2:
	UF : 1, UT : 1,
	J1=    90.000 deg,	J2=   -90.000 deg
};
P[580]{
   GP1:
	UF : 1, UT : 1,		CONFIG : 'N U T, 0, 0, 0',
	X =  1548.450  mm,	Y =   -29.796  mm,	Z =   -15.951  mm,
	W =    36.729 deg,	P =    28.085 deg,	R =   -43.976 deg
   GP2:
	UF : 1, UT : 1,
	J1=    90.000 deg,	J2=   -90.000 deg
};
P[581]{
   GP1:
	UF : 1, UT : 1,		CONFIG : 'N U T, 0, 0, 0',
	X =  2158.527  mm,	Y =  -106.081  mm,	Z =    42.026  mm,
	W =    44.885 deg,	P =     3.628 deg,	R =    -3.635 deg
   GP2:
	UF : 1, UT : 1,
	J1=    90.000 deg,	J2=   -90.000 deg
};
P[582]{
   GP1:
	UF : 1, UT : 1,		CONFIG : 'N U T, 0, 0, 0',
	X =  1541.843  mm,	Y =   -26.526  mm,	Z =   -17.050  mm,
	W =    36.730 deg,	P =    28.085 deg,	R =   -43.977 deg
   GP2:
	UF : 1, UT : 1,
	J1=    90.000 deg,	J2=   -90.000 deg
};
P[583]{
   GP1:
	UF : 1, UT : 1,		CONFIG : 'N U T, 0, 0, 0',
	X =  2359.776  mm,	Y =   167.003  mm,	Z =    -8.816  mm,
	W =    38.121 deg,	P =   -25.966 deg,	R =    27.297 deg
   GP2:
	UF : 1, UT : 1,
	J1=    90.000 deg,	J2=   -90.000 deg
};
P[584]{
   GP1:
	UF : 1, UT : 1,		CONFIG : 'N U T, 0, 0, 0',
	X =  2406.274  mm,	Y =   166.697  mm,	Z =    -9.876  mm,
	W =    38.121 deg,	P =   -25.966 deg,	R =    27.297 deg
   GP2:
	UF : 1, UT : 1,
	J1=    90.000 deg,	J2=   -90.000 deg
};
P[585]{
   GP1:
	UF : 1, UT : 1,		CONFIG : 'N U T, 0, 0, 0',
	X =  2060.197  mm,	Y =  -106.080  mm,	Z =    42.026  mm,
	W =    44.885 deg,	P =     3.628 deg,	R =    -3.635 deg
   GP2:
	UF : 1, UT : 1,
	J1=    90.000 deg,	J2=   -90.000 deg
};
P[586]{
   GP1:
	UF : 1, UT : 1,		CONFIG : 'N U T, 0, 0, 0',
	X =  2420.811  mm,	Y =   162.873  mm,	Z =    -7.347  mm,
	W =     9.855 deg,	P =   -38.956 deg,	R =    41.531 deg
   GP2:
	UF : 1, UT : 1,
	J1=    89.988 deg,	J2=   -90.001 deg
};
P[587]{
   GP1:
	UF : 1, UT : 1,		CONFIG : 'N U T, 0, 0, 0',
	X =  1671.414  mm,	Y =   189.046  mm,	Z =   -15.712  mm,
	W =   -36.940 deg,	P =    22.774 deg,	R =   -15.979 deg
   GP2:
	UF : 1, UT : 1,
	J1=    90.000 deg,	J2=   -90.000 deg
};
P[588]{
   GP1:
	UF : 1, UT : 1,		CONFIG : 'N U T, 0, 0, 0',
	X =  1704.592  mm,	Y =   193.463  mm,	Z =   -14.287  mm,
	W =   -36.936 deg,	P =    22.774 deg,	R =    39.322 deg
   GP2:
	UF : 1, UT : 1,
	J1=    90.000 deg,	J2=   -90.000 deg
};
P[589]{
   GP1:
	UF : 1, UT : 1,		CONFIG : 'N U T, 0, 0, 0',
	X =  1890.253  mm,	Y =  -197.333  mm,	Z =   104.046  mm,
	W =    40.690 deg,	P =   -21.162 deg,	R =    -6.795 deg
   GP2:
	UF : 1, UT : 1,
	J1=    90.000 deg,	J2=   -90.000 deg
};
P[590]{
   GP1:
	UF : 1, UT : 1,		CONFIG : 'N U T, 0, 0, 0',
	X =  1890.254  mm,	Y =  -197.333  mm,	Z =   104.046  mm,
	W =   -33.760 deg,	P =   -16.746 deg,	R =    41.760 deg
   GP2:
	UF : 1, UT : 1,
	J1=    90.000 deg,	J2=   -90.000 deg
};
P[591]{
   GP1:
	UF : 1, UT : 1,		CONFIG : 'N U T, 0, 0, 0',
	X =  2024.254  mm,	Y =  -116.333  mm,	Z =   104.046  mm,
	W =   -36.632 deg,	P =    -7.222 deg,	R =    55.482 deg
   GP2:
	UF : 1, UT : 1,
	J1=    90.000 deg,	J2=   -90.000 deg
};
P[592]{
   GP1:
	UF : 1, UT : 1,		CONFIG : 'N U T, 0, 0, 0',
	X =  1976.573  mm,	Y =   191.971  mm,	Z =   -16.183  mm,
	W =   -36.940 deg,	P =    22.774 deg,	R =    39.323 deg
   GP2:
	UF : 1, UT : 1,
	J1=    90.000 deg,	J2=   -90.000 deg
};
P[593]{
   GP1:
	UF : 1, UT : 1,		CONFIG : 'N U T, 0, 0, 0',
	X =  1990.474  mm,	Y =   191.565  mm,	Z =   -18.105  mm,
	W =   -40.749 deg,	P =    13.396 deg,	R =    62.815 deg
   GP2:
	UF : 1, UT : 1,
	J1=    90.000 deg,	J2=   -90.000 deg
};
P[594]{
   GP1:
	UF : 1, UT : 1,		CONFIG : 'N U T, 0, 0, 0',
	X =  2392.053  mm,	Y =    84.549  mm,	Z =   -21.907  mm,
	W =   -47.015 deg,	P =     6.660 deg,	R =   -51.412 deg
   GP2:
	UF : 1, UT : 1,
	J1=    83.000 deg,	J2=   -90.000 deg
};
P[595]{
   GP1:
	UF : 1, UT : 1,		CONFIG : 'N U T, 0, 0, 0',
	X =  2056.301  mm,	Y =   -98.366  mm,	Z =    49.506  mm,
	W =   -42.382 deg,	P =     2.305 deg,	R =   105.198 deg
   GP2:
	UF : 1, UT : 1,
	J1=    90.000 deg,	J2=   -90.000 deg
};
P[596]{
   GP1:
	UF : 1, UT : 1,		CONFIG : 'N U T, 0, 0, 1',
	X =  1663.323  mm,	Y =  -387.368  mm,	Z =   408.939  mm,
	W =   -27.547 deg,	P =    30.353 deg,	R =   152.229 deg
   GP2:
	UF : 1, UT : 1,
	J1=    90.000 deg,	J2=   -90.000 deg
};
P[597]{
   GP1:
	UF : 1, UT : 1,		CONFIG : 'N U T, 0, 0, 1',
	X =  1656.330  mm,	Y =  -300.541  mm,	Z =  1123.310  mm,
	W =    -9.281 deg,	P =    48.130 deg,	R =  -175.012 deg
   GP2:
	UF : 1, UT : 1,
	J1=    90.000 deg,	J2=   -90.000 deg
};
P[598]{
   GP1:
	UF : 1, UT : 1,		CONFIG : 'N U T, 0, 0, 1',
	X =  2106.086  mm,	Y =  -147.825  mm,	Z =   986.847  mm,
